LIN {X 0,Y 509.393,Z 1059.05,A -85,B 0,C 180,E1 -5481.271,E2 -5481.271} C_VEL
LIN {X 0,Y 509.308,Z 1064.075,A -85,B 0,C 180,E1 -5482.866,E2 -5482.866} C_VEL
LIN {X 0,Y 509.215,Z 1068.022,A -85,B 0,C 180,E1 -5484.456,E2 -5484.456} C_VEL
LIN {X 0,Y 509.196,Z 1070.928,A -85,B 0,C 180,E1 -5486.043,E2 -5486.043} C_VEL
LIN {X 0,Y 509.184,Z 1072.082,A -85,B 0,C 180,E1 -5486.835,E2 -5486.835} C_VEL
LIN {X 0,Y 509.107,Z 1073.515,A -85,B 0,C 180,E1 -5488.418,E2 -5488.418} C_VEL
LIN {X 0,Y 509.061,Z 1074,A -85,B 0,C 180,E1 -5490,E2 -5490} C_VEL
LIN {X 0,Y 509.107,Z 1073.515,A -85,B 0,C 180,E1 -5491.582,E2 -5491.582} C_VEL
LIN {X 0,Y 509.184,Z 1072.082,A -85,B 0,C 180,E1 -5493.165,E2 -5493.165} C_VEL
LIN {X 0,Y 509.142,Z 1069.669,A -85,B 0,C 180,E1 -5494.751,E2 -5494.751} C_VEL
LIN {X 0,Y 509.264,Z 1065.849,A -85,B 0,C 180,E1 -5496.476,E2 -5496.476} C_VEL
LIN {X 0,Y 509.332,Z 1061.713,A -85,B 0,C 180,E1 -5497.931,E2 -5497.931} C_VEL
LIN {X 0,Y 509.421,Z 1056.051,A -85,B 0,C 180,E1 -5499.529,E2 -5499.529} C_VEL
LIN {X 0,Y 509.628,Z 1051.052,A -85,B 0,C 180,E1 -5500.729,E2 -5500.729} C_VEL
LIN {X 0,Y 509.913,Z 1044.199,A -85,B 0,C 180,E1 -5502.133,E2 -5502.133} C_VEL
LIN {X 0,Y 510.2,Z 1036.178,A -85,B 0,C 180,E1 -5503.543,E2 -5503.543} C_VEL
LIN {X 0,Y 510.601,Z 1028.274,A -85,B 0,C 180,E1 -5504.752,E2 -5504.752} C_VEL
LIN {X 0,Y 511.042,Z 1019.227,A -85,B 0,C 180,E1 -5505.964,E2 -5505.964} C_VEL
LIN {X 0,Y 511.563,Z 1008.82,A -85,B 0,C 180,E1 -5507.179,E2 -5507.179} C_VEL
LIN {X 0,Y 512.103,Z 998.917,A -85,B 0,C 180,E1 -5508.192,E2 -5508.192} C_VEL
LIN {X 0,Y 512.69,Z 989.263,A -85,B 0,C 180,E1 -5509.065,E2 -5509.065} C_VEL
LIN {X 0,Y 513.308,Z 977.141,A -85,B 0,C 180,E1 -5510.016,E2 -5510.016} C_VEL
LIN {X 0,Y 513.876,Z 965.105,A -85,B 0,C 180,E1 -5510.829,E2 -5510.829} C_VEL
LIN {X 0,Y 514.531,Z 952.779,A -85,B 0,C 180,E1 -5511.535,E2 -5511.535} C_VEL
LIN {X 0,Y 515.092,Z 939.627,A -85,B 0,C 180,E1 -5512.169,E2 -5512.169} C_VEL
LIN {X 0,Y 515.587,Z 926.791,A -85,B 0,C 180,E1 -5512.674,E2 -5512.674} C_VEL
LIN {X 0,Y 515.947,Z 913.864,A -85,B 0,C 180,E1 -5513.081,E2 -5513.081} C_VEL
LIN {X 0,Y 516.291,Z 901.026,A -85,B 0,C 180,E1 -5513.383,E2 -5513.383} C_VEL
LIN {X 0,Y 516.696,Z 874.989,A -85,B 0,C 180,E1 -5513.789,E2 -5513.789} C_VEL
LIN {X 0,Y 518.063,Z 714.987,A -85,B 0,C 180,E1 -5516.115,E2 -5516.115} C_VEL
LIN {X 0,Y 513.214,Z 695.236,A -85,B 0,C 180,E1 -5516.696,E2 -5516.696} C_VEL
LIN {X 0,Y 514.044,Z 674.695,A -85,B 0,C 180,E1 -5519.709,E2 -5519.709} C_VEL
LIN {X 0,Y 513.889,Z 670.977,A -85,B 0,C 180,E1 -5520.284,E2 -5520.284} C_VEL
LIN {X 0,Y 509.916,Z 655.134,A -85,B 0,C 180,E1 -5523.033,E2 -5523.033} C_VEL
LIN {X 0,Y 509.867,Z 654.796,A -85,B 0,C 180,E1 -5523.178,E2 -5523.178} C_VEL
LIN {X 0,Y 509.83,Z 654.762,A -85,B 0,C 180,E1 -5526.352,E2 -5526.352} C_VEL
LIN {X 0,Y 509.83,Z 654.793,A -85,B 0,C 180,E1 -5529.47,E2 -5529.47} C_VEL
LIN {X 0,Y 509.842,Z 654.786,A -85,B 0,C 180,E1 -5532.487,E2 -5532.487} C_VEL
LIN {X 0,Y 509.85,Z 654.781,A -85,B 0,C 180,E1 -5535.331,E2 -5535.331} C_VEL
LIN {X 0,Y 509.866,Z 654.772,A -85,B 0,C 180,E1 -5538.576,E2 -5538.576} C_VEL
LIN {X 0,Y 509.849,Z 654.791,A -85,B 0,C 180,E1 -5541.785,E2 -5541.785} C_VEL
LIN {X 0,Y 509.839,Z 654.777,A -85,B 0,C 180,E1 -5544.623,E2 -5544.623} C_VEL
LIN {X 0,Y 509.858,Z 654.785,A -85,B 0,C 180,E1 -5547.481,E2 -5547.481} C_VEL
LIN {X 0,Y 509.873,Z 654.766,A -85,B 0,C 180,E1 -5550.268,E2 -5550.268} C_VEL
LIN {X 0,Y 509.878,Z 654.775,A -85,B 0,C 180,E1 -5552.944,E2 -5552.944} C_VEL
LIN {X 0,Y 509.86,Z 654.783,A -85,B 0,C 180,E1 -5555.573,E2 -5555.573} C_VEL
LIN {X 0,Y 509.813,Z 654.787,A -85,B 0,C 180,E1 -5558.148,E2 -5558.148} C_VEL
LIN {X 0,Y 509.855,Z 654.787,A -85,B 0,C 180,E1 -5560.681,E2 -5560.681} C_VEL
LIN {X 0,Y 509.877,Z 654.782,A -85,B 0,C 180,E1 -5563.174,E2 -5563.174} C_VEL
LIN {X 0,Y 509.854,Z 654.781,A -85,B 0,C 180,E1 -5565.634,E2 -5565.634} C_VEL
LIN {X 0,Y 509.919,Z 654.781,A -85,B 0,C 180,E1 -5568.875,E2 -5568.875} C_VEL
LIN {X 0,Y 509.941,Z 654.764,A -85,B 0,C 180,E1 -5572.078,E2 -5572.078} C_VEL
LIN {X 0,Y 510.001,Z 654.764,A -85,B 0,C 180,E1 -5574.464,E2 -5574.464} C_VEL
LIN {X 0,Y 510.045,Z 654.76,A -85,B 0,C 180,E1 -5577.631,E2 -5577.631} C_VEL
LIN {X 0,Y 510.056,Z 654.759,A -85,B 0,C 180,E1 -5580.789,E2 -5580.789} C_VEL
LIN {X 0,Y 509.95,Z 654.767,A -85,B 0,C 180,E1 -5583.16,E2 -5583.16} C_VEL
LIN {X 0,Y 509.972,Z 654.766,A -85,B 0,C 180,E1 -5586.329,E2 -5586.329} C_VEL
LIN {X 0,Y 509.908,Z 654.773,A -85,B 0,C 180,E1 -5588.72,E2 -5588.72} C_VEL
LIN {X 0,Y 509.893,Z 654.779,A -85,B 0,C 180,E1 -5591.932,E2 -5591.932} C_VEL
LIN {X 0,Y 509.882,Z 654.779,A -85,B 0,C 180,E1 -5595.242,E2 -5595.242} C_VEL
LIN {X 0,Y 509.877,Z 654.781,A -85,B 0,C 180,E1 -5598.001,E2 -5598.001} C_VEL
LIN {X 0,Y 509.848,Z 654.782,A -85,B 0,C 180,E1 -5601.001,E2 -5601.001} C_VEL
LIN {X 0,Y 509.841,Z 654.783,A -85,B 0,C 180,E1 -5603.563,E2 -5603.563} C_VEL
LIN {X 0,Y 509.902,Z 654.777,A -85,B 0,C 180,E1 -5606.379,E2 -5606.379} C_VEL
LIN {X 0,Y 509.875,Z 654.766,A -85,B 0,C 180,E1 -5608.844,E2 -5608.844} C_VEL
LIN {X 0,Y 509.816,Z 654.787,A -85,B 0,C 180,E1 -5611.59,E2 -5611.59} C_VEL
LIN {X 0,Y 509.845,Z 654.787,A -85,B 0,C 180,E1 -5614.413,E2 -5614.413} C_VEL
LIN {X 0,Y 509.809,Z 654.788,A -85,B 0,C 180,E1 -5617.341,E2 -5617.341} C_VEL
LIN {X 0,Y 509.854,Z 654.785,A -85,B 0,C 180,E1 -5620.38,E2 -5620.38} C_VEL
LIN {X 0,Y 509.833,Z 654.795,A -85,B 0,C 180,E1 -5623.065,E2 -5623.065} C_VEL
LIN {X 0,Y 509.822,Z 654.789,A -85,B 0,C 180,E1 -5625.793,E2 -5625.793} C_VEL
LIN {X 0,Y 509.857,Z 654.784,A -85,B 0,C 180,E1 -5628.576,E2 -5628.576} C_VEL
LIN {X 0,Y 509.844,Z 654.79,A -85,B 0,C 180,E1 -5631.787,E2 -5631.787} C_VEL
LIN {X 0,Y 509.825,Z 654.793,A -85,B 0,C 180,E1 -5633.744,E2 -5633.744} C_VEL
LIN {X 0,Y 509.159,Z 654.872,A -85,B 0,C 180,E1 -5634.404,E2 -5634.404} C_VEL
LIN {X 0,Y 506.341,Z 655.229,A -85,B 0,C 180,E1 -5635.476,E2 -5635.476} C_VEL
LIN {X 0,Y 503.947,Z 655.524,A -85,B 0,C 180,E1 -5636.339,E2 -5636.339} C_VEL
LIN {X 0,Y 502.899,Z 655.652,A -85,B 0,C 180,E1 -5637.006,E2 -5637.006} C_VEL
LIN {X 0,Y 502.802,Z 655.664,A -85,B 0,C 180,E1 -5637.231,E2 -5637.231} C_VEL
LIN {X 0,Y 502.824,Z 655.666,A -85,B 0,C 180,E1 -5640.062,E2 -5640.062} C_VEL
LIN {X 0,Y 502.828,Z 655.661,A -85,B 0,C 180,E1 -5642.534,E2 -5642.534} C_VEL
LIN {X 0,Y 502.823,Z 655.661,A -85,B 0,C 180,E1 -5645.299,E2 -5645.299} C_VEL
LIN {X 0,Y 502.78,Z 655.672,A -85,B 0,C 180,E1 -5647.827,E2 -5647.827} C_VEL
LIN {X 0,Y 502.82,Z 655.666,A -85,B 0,C 180,E1 -5650.401,E2 -5650.401} C_VEL
LIN {X 0,Y 502.829,Z 655.661,A -85,B 0,C 180,E1 -5652.932,E2 -5652.932} C_VEL
LIN {X 0,Y 502.841,Z 655.659,A -85,B 0,C 180,E1 -5655.429,E2 -5655.429} C_VEL
LIN {X 0,Y 502.873,Z 655.66,A -85,B 0,C 180,E1 -5658.717,E2 -5658.717} C_VEL
LIN {X 0,Y 502.898,Z 655.652,A -85,B 0,C 180,E1 -5661.967,E2 -5661.967} C_VEL
LIN {X 0,Y 502.934,Z 655.65,A -85,B 0,C 180,E1 -5664.387,E2 -5664.387} C_VEL
LIN {X 0,Y 503.021,Z 655.637,A -85,B 0,C 180,E1 -5667.598,E2 -5667.598} C_VEL
LIN {X 0,Y 503.024,Z 655.637,A -85,B 0,C 180,E1 -5670,E2 -5670} C_VEL
LIN {X 0,Y 503.021,Z 655.637,A -85,B 0,C 180,E1 -5672.402,E2 -5672.402} C_VEL
LIN {X 0,Y 502.934,Z 655.65,A -85,B 0,C 180,E1 -5675.613,E2 -5675.613} C_VEL
LIN {X 0,Y 502.898,Z 655.652,A -85,B 0,C 180,E1 -5678.033,E2 -5678.033} C_VEL
LIN {X 0,Y 502.873,Z 655.66,A -85,B 0,C 180,E1 -5681.283,E2 -5681.283} C_VEL
LIN {X 0,Y 502.841,Z 655.659,A -85,B 0,C 180,E1 -5684.571,E2 -5684.571} C_VEL
LIN {X 0,Y 502.857,Z 655.661,A -85,B 0,C 180,E1 -5687.907,E2 -5687.907} C_VEL
LIN {X 0,Y 502.823,Z 655.661,A -85,B 0,C 180,E1 -5690.536,E2 -5690.536} C_VEL
LIN {X 0,Y 502.792,Z 655.665,A -85,B 0,C 180,E1 -5693.04,E2 -5693.04} C_VEL
LIN {X 0,Y 502.835,Z 655.663,A -85,B 0,C 180,E1 -5695.675,E2 -5695.675} C_VEL
LIN {X 0,Y 502.836,Z 655.664,A -85,B 0,C 180,E1 -5698.372,E2 -5698.372} C_VEL
LIN {X 0,Y 502.791,Z 655.665,A -85,B 0,C 180,E1 -5701.499,E2 -5701.499} C_VEL
LIN {X 0,Y 502.799,Z 655.67,A -85,B 0,C 180,E1 -5704.444,E2 -5704.444} C_VEL
LIN {X 0,Y 502.774,Z 655.667,A -85,B 0,C 180,E1 -5707.178,E2 -5707.178} C_VEL
LIN {X 0,Y 502.814,Z 655.662,A -85,B 0,C 180,E1 -5710.011,E2 -5710.011} C_VEL
LIN {X 0,Y 502.764,Z 655.67,A -85,B 0,C 180,E1 -5713.231,E2 -5713.231} C_VEL
LIN {X 0,Y 502.781,Z 655.665,A -85,B 0,C 180,E1 -5715.661,E2 -5715.661} C_VEL
LIN {X 0,Y 502.83,Z 655.659,A -85,B 0,C 180,E1 -5717.865,E2 -5717.865} C_VEL
LIN {X 0,Y 502.812,Z 655.668,A -85,B 0,C 180,E1 -5721.026,E2 -5721.026} C_VEL
LIN {X 0,Y 502.775,Z 655.648,A -85,B 0,C 180,E1 -5724.167,E2 -5724.167} C_VEL
LIN {X 0,Y 502.823,Z 655.662,A -85,B 0,C 180,E1 -5726.993,E2 -5726.993} C_VEL
LIN {X 0,Y 502.82,Z 655.646,A -85,B 0,C 180,E1 -5730.061,E2 -5730.061} C_VEL
LIN {X 0,Y 502.825,Z 655.647,A -85,B 0,C 180,E1 -5732.533,E2 -5732.533} C_VEL
LIN {X 0,Y 502.82,Z 655.663,A -85,B 0,C 180,E1 -5735.298,E2 -5735.298} C_VEL
LIN {X 0,Y 502.809,Z 655.662,A -85,B 0,C 180,E1 -5737.828,E2 -5737.828} C_VEL
LIN {X 0,Y 502.814,Z 655.661,A -85,B 0,C 180,E1 -5740.4,E2 -5740.4} C_VEL
LIN {X 0,Y 502.825,Z 655.654,A -85,B 0,C 180,E1 -5742.932,E2 -5742.932} C_VEL
LIN {X 0,Y 502.834,Z 655.658,A -85,B 0,C 180,E1 -5745.429,E2 -5745.429} C_VEL
LIN {X 0,Y 502.87,Z 655.654,A -85,B 0,C 180,E1 -5748.717,E2 -5748.717} C_VEL
LIN {X 0,Y 502.891,Z 655.65,A -85,B 0,C 180,E1 -5751.967,E2 -5751.967} C_VEL
LIN {X 0,Y 502.952,Z 655.649,A -85,B 0,C 180,E1 -5754.387,E2 -5754.387} C_VEL
LIN {X 0,Y 503.015,Z 655.627,A -85,B 0,C 180,E1 -5757.598,E2 -5757.598} C_VEL
LIN {X 0,Y 503.015,Z 655.636,A -85,B 0,C 180,E1 -5760,E2 -5760} C_VEL
LIN {X 0,Y 503.015,Z 655.636,A -85,B 0,C 180,E1 -5762.402,E2 -5762.402} C_VEL
LIN {X 0,Y 502.952,Z 655.642,A -85,B 0,C 180,E1 -5765.614,E2 -5765.614} C_VEL
LIN {X 0,Y 502.892,Z 655.641,A -85,B 0,C 180,E1 -5768.034,E2 -5768.034} C_VEL
LIN {X 0,Y 502.887,Z 655.653,A -85,B 0,C 180,E1 -5771.283,E2 -5771.283} C_VEL
LIN {X 0,Y 502.834,Z 655.656,A -85,B 0,C 180,E1 -5774.571,E2 -5774.571} C_VEL
LIN {X 0,Y 502.852,Z 655.653,A -85,B 0,C 180,E1 -5777.907,E2 -5777.907} C_VEL
LIN {X 0,Y 502.818,Z 655.659,A -85,B 0,C 180,E1 -5780.537,E2 -5780.537} C_VEL
LIN {X 0,Y 502.787,Z 655.659,A -85,B 0,C 180,E1 -5783.041,E2 -5783.041} C_VEL
LIN {X 0,Y 502.832,Z 655.662,A -85,B 0,C 180,E1 -5785.676,E2 -5785.676} C_VEL
LIN {X 0,Y 502.833,Z 655.635,A -85,B 0,C 180,E1 -5788.373,E2 -5788.373} C_VEL
LIN {X 0,Y 502.789,Z 655.662,A -85,B 0,C 180,E1 -5791.5,E2 -5791.5} C_VEL
LIN {X 0,Y 502.799,Z 655.656,A -85,B 0,C 180,E1 -5794.446,E2 -5794.446} C_VEL
LIN {X 0,Y 502.774,Z 655.661,A -85,B 0,C 180,E1 -5797.179,E2 -5797.179} C_VEL
LIN {X 0,Y 502.828,Z 655.661,A -85,B 0,C 180,E1 -5800.011,E2 -5800.011} C_VEL
LIN {X 0,Y 502.82,Z 655.656,A -85,B 0,C 180,E1 -5802.203,E2 -5802.203} C_VEL
LIN {X 0,Y 502.794,Z 655.653,A -85,B 0,C 180,E1 -5805.469,E2 -5805.469} C_VEL
LIN {X 0,Y 502.824,Z 655.662,A -85,B 0,C 180,E1 -5807.865,E2 -5807.865} C_VEL
LIN {X 0,Y 502.797,Z 655.666,A -85,B 0,C 180,E1 -5811.025,E2 -5811.025} C_VEL
LIN {X 0,Y 502.78,Z 655.642,A -85,B 0,C 180,E1 -5814.168,E2 -5814.168} C_VEL
LIN {X 0,Y 502.851,Z 655.759,A -85,B 0,C 180,E1 -5816.559,E2 -5816.559} C_VEL
LIN {X 0,Y 506.42,Z 669.991,A -85,B 0,C 180,E1 -5819.105,E2 -5819.105} C_VEL
LIN {X 0,Y 507.298,Z 674.677,A -85,B 0,C 180,E1 -5819.886,E2 -5819.886} C_VEL
LIN {X 0,Y 506.412,Z 694.461,A -85,B 0,C 180,E1 -5822.866,E2 -5822.866} C_VEL
LIN {X 0,Y 506.693,Z 696.204,A -85,B 0,C 180,E1 -5822.965,E2 -5822.965} C_VEL
LIN {X 0,Y 511.701,Z 716.956,A -85,B 0,C 180,E1 -5823.569,E2 -5823.569} C_VEL
LIN {X 0,Y 509.898,Z 896.602,A -85,B 0,C 180,E1 -5826.225,E2 -5826.225} C_VEL
LIN {X 0,Y 509.497,Z 909.739,A -85,B 0,C 180,E1 -5826.502,E2 -5826.502} C_VEL
LIN {X 0,Y 509.137,Z 922.851,A -85,B 0,C 180,E1 -5826.888,E2 -5826.888} C_VEL
LIN {X 0,Y 508.613,Z 935.231,A -85,B 0,C 180,E1 -5827.346,E2 -5827.346} C_VEL
LIN {X 0,Y 508.097,Z 948.012,A -85,B 0,C 180,E1 -5827.932,E2 -5827.932} C_VEL
LIN {X 0,Y 507.494,Z 959.929,A -85,B 0,C 180,E1 -5828.581,E2 -5828.581} C_VEL
LIN {X 0,Y 506.819,Z 972.616,A -85,B 0,C 180,E1 -5829.399,E2 -5829.399} C_VEL
LIN {X 0,Y 506.202,Z 983.621,A -85,B 0,C 180,E1 -5830.22,E2 -5830.22} C_VEL
LIN {X 0,Y 505.486,Z 995.193,A -85,B 0,C 180,E1 -5831.215,E2 -5831.215} C_VEL
LIN {X 0,Y 504.949,Z 1004.935,A -85,B 0,C 180,E1 -5832.17,E2 -5832.17} C_VEL
LIN {X 0,Y 504.419,Z 1014.211,A -85,B 0,C 180,E1 -5833.196,E2 -5833.196} C_VEL
LIN {X 0,Y 503.865,Z 1023.624,A -85,B 0,C 180,E1 -5834.385,E2 -5834.385} C_VEL
LIN {X 0,Y 503.377,Z 1032.363,A -85,B 0,C 180,E1 -5835.652,E2 -5835.652} C_VEL
LIN {X 0,Y 502.964,Z 1040.89,A -85,B 0,C 180,E1 -5837.082,E2 -5837.082} C_VEL
LIN {X 0,Y 502.721,Z 1048.049,A -85,B 0,C 180,E1 -5838.475,E2 -5838.475} C_VEL
LIN {X 0,Y 502.431,Z 1054.443,A -85,B 0,C 180,E1 -5839.93,E2 -5839.93} C_VEL
LIN {X 0,Y 502.309,Z 1059.044,A -85,B 0,C 180,E1 -5841.147,E2 -5841.147} C_VEL
LIN {X 0,Y 502.231,Z 1064.071,A -85,B 0,C 180,E1 -5842.765,E2 -5842.765} C_VEL
LIN {X 0,Y 502.132,Z 1068.016,A -85,B 0,C 180,E1 -5844.378,E2 -5844.378} C_VEL
LIN {X 0,Y 502.09,Z 1070.924,A -85,B 0,C 180,E1 -5845.987,E2 -5845.987} C_VEL
LIN {X 0,Y 502.103,Z 1072.082,A -85,B 0,C 180,E1 -5846.791,E2 -5846.791} C_VEL
LIN {X 0,Y 502.03,Z 1073.518,A -85,B 0,C 180,E1 -5848.396,E2 -5848.396} C_VEL
LIN {X 0,Y 501.975,Z 1074,A -85,B 0,C 180,E1 -5850,E2 -5850} C_VEL
LIN {X 0,Y 502.03,Z 1073.518,A -85,B 0,C 180,E1 -5851.604,E2 -5851.604} C_VEL
LIN {X 0,Y 502.103,Z 1072.082,A -85,B 0,C 180,E1 -5853.209,E2 -5853.209} C_VEL
LIN {X 0,Y 502.061,Z 1069.666,A -85,B 0,C 180,E1 -5854.818,E2 -5854.818} C_VEL
LIN {X 0,Y 502.194,Z 1065.145,A -85,B 0,C 180,E1 -5856.831,E2 -5856.831} C_VEL
LIN {X 0,Y 502.248,Z 1061.707,A -85,B 0,C 180,E1 -5858.044,E2 -5858.044} C_VEL
LIN {X 0,Y 502.354,Z 1056.046,A -85,B 0,C 180,E1 -5859.664,E2 -5859.664} C_VEL
LIN {X 0,Y 502.585,Z 1051.046,A -85,B 0,C 180,E1 -5860.881,E2 -5860.881} C_VEL
LIN {X 0,Y 502.878,Z 1044.193,A -85,B 0,C 180,E1 -5862.305,E2 -5862.305} C_VEL
LIN {X 0,Y 503.2,Z 1036.171,A -85,B 0,C 180,E1 -5863.735,E2 -5863.735} C_VEL
LIN {X 0,Y 503.67,Z 1028.267,A -85,B 0,C 180,E1 -5864.959,E2 -5864.959} C_VEL
LIN {X 0,Y 504.152,Z 1019.22,A -85,B 0,C 180,E1 -5866.188,E2 -5866.188} C_VEL
LIN {X 0,Y 504.599,Z 1010.657,A -85,B 0,C 180,E1 -5867.215,E2 -5867.215} C_VEL
LIN {X 0,Y 505.266,Z 998.783,A -85,B 0,C 180,E1 -5868.447,E2 -5868.447} C_VEL
LIN {X 0,Y 505.944,Z 988.463,A -85,B 0,C 180,E1 -5869.381,E2 -5869.381} C_VEL
LIN {X 0,Y 506.575,Z 976.934,A -85,B 0,C 180,E1 -5870.294,E2 -5870.294} C_VEL
LIN {X 0,Y 507.177,Z 964.897,A -85,B 0,C 180,E1 -5871.117,E2 -5871.117} C_VEL
LIN {X 0,Y 507.851,Z 953.134,A -85,B 0,C 180,E1 -5871.803,E2 -5871.803} C_VEL
LIN {X 0,Y 508.465,Z 939.42,A -85,B 0,C 180,E1 -5872.473,E2 -5872.473} C_VEL
LIN {X 0,Y 509.013,Z 926.584,A -85,B 0,C 180,E1 -5872.984,E2 -5872.984} C_VEL
LIN {X 0,Y 509.39,Z 913.658,A -85,B 0,C 180,E1 -5873.396,E2 -5873.396} C_VEL
LIN {X 0,Y 509.765,Z 900.82,A -85,B 0,C 180,E1 -5873.701,E2 -5873.701} C_VEL
LIN {X 0,Y 510.216,Z 874.784,A -85,B 0,C 180,E1 -5874.11,E2 -5874.11} C_VEL
LIN {X 0,Y 511.593,Z 715.983,A -85,B 0,C 180,E1 -5876.452,E2 -5876.452} C_VEL
LIN {X 0,Y 506.442,Z 694.904,A -85,B 0,C 180,E1 -5877.087,E2 -5877.087} C_VEL
LIN {X 0,Y 507.301,Z 675.964,A -85,B 0,C 180,E1 -5879.915,E2 -5879.915} C_VEL
LIN {X 0,Y 506.98,Z 672.28,A -85,B 0,C 180,E1 -5880.504,E2 -5880.504} C_VEL
LIN {X 0,Y 502.881,Z 655.971,A -85,B 0,C 180,E1 -5883.385,E2 -5883.385} C_VEL
LIN {X 0,Y 502.823,Z 655.687,A -85,B 0,C 180,E1 -5883.509,E2 -5883.509} C_VEL
LIN {X 0,Y 502.778,Z 655.641,A -85,B 0,C 180,E1 -5885.95,E2 -5885.95} C_VEL
LIN {X 0,Y 502.797,Z 655.666,A -85,B 0,C 180,E1 -5888.975,E2 -5888.975} C_VEL
LIN {X 0,Y 502.824,Z 655.662,A -85,B 0,C 180,E1 -5892.135,E2 -5892.135} C_VEL
LIN {X 0,Y 502.795,Z 655.662,A -85,B 0,C 180,E1 -5895.467,E2 -5895.467} C_VEL
LIN {X 0,Y 502.832,Z 655.654,A -85,B 0,C 180,E1 -5897.864,E2 -5897.864} C_VEL
LIN {X 0,Y 502.815,Z 655.661,A -85,B 0,C 180,E1 -5901.025,E2 -5901.025} C_VEL
LIN {X 0,Y 502.778,Z 655.656,A -85,B 0,C 180,E1 -5904.166,E2 -5904.166} C_VEL
LIN {X 0,Y 502.825,Z 655.659,A -85,B 0,C 180,E1 -5906.992,E2 -5906.992} C_VEL
LIN {X 0,Y 502.822,Z 655.647,A -85,B 0,C 180,E1 -5910.061,E2 -5910.061} C_VEL
LIN {X 0,Y 502.826,Z 655.651,A -85,B 0,C 180,E1 -5912.533,E2 -5912.533} C_VEL
LIN {X 0,Y 502.819,Z 655.66,A -85,B 0,C 180,E1 -5915.298,E2 -5915.298} C_VEL
LIN {X 0,Y 502.775,Z 655.66,A -85,B 0,C 180,E1 -5917.826,E2 -5917.826} C_VEL
LIN {X 0,Y 502.816,Z 655.667,A -85,B 0,C 180,E1 -5920.4,E2 -5920.4} C_VEL
LIN {X 0,Y 502.827,Z 655.663,A -85,B 0,C 180,E1 -5922.931,E2 -5922.931} C_VEL
LIN {X 0,Y 502.834,Z 655.657,A -85,B 0,C 180,E1 -5925.429,E2 -5925.429} C_VEL
LIN {X 0,Y 502.887,Z 655.654,A -85,B 0,C 180,E1 -5928.717,E2 -5928.717} C_VEL
LIN {X 0,Y 502.892,Z 655.641,A -85,B 0,C 180,E1 -5931.966,E2 -5931.966} C_VEL
LIN {X 0,Y 502.952,Z 655.642,A -85,B 0,C 180,E1 -5934.386,E2 -5934.386} C_VEL
LIN {X 0,Y 503.015,Z 655.636,A -85,B 0,C 180,E1 -5937.598,E2 -5937.598} C_VEL
LIN {X 0,Y 503.015,Z 655.635,A -85,B 0,C 180,E1 -5940,E2 -5940} C_VEL
LIN {X 0,Y 503.015,Z 655.626,A -85,B 0,C 180,E1 -5942.402,E2 -5942.402} C_VEL
LIN {X 0,Y 502.952,Z 655.65,A -85,B 0,C 180,E1 -5945.613,E2 -5945.613} C_VEL
LIN {X 0,Y 502.891,Z 655.651,A -85,B 0,C 180,E1 -5948.033,E2 -5948.033} C_VEL
LIN {X 0,Y 502.87,Z 655.654,A -85,B 0,C 180,E1 -5951.283,E2 -5951.283} C_VEL
LIN {X 0,Y 502.834,Z 655.658,A -85,B 0,C 180,E1 -5954.571,E2 -5954.571} C_VEL
LIN {X 0,Y 502.85,Z 655.655,A -85,B 0,C 180,E1 -5957.907,E2 -5957.907} C_VEL
LIN {X 0,Y 502.819,Z 655.662,A -85,B 0,C 180,E1 -5960.537,E2 -5960.537} C_VEL
LIN {X 0,Y 502.804,Z 655.66,A -85,B 0,C 180,E1 -5963.04,E2 -5963.04} C_VEL
LIN {X 0,Y 502.831,Z 655.658,A -85,B 0,C 180,E1 -5965.676,E2 -5965.676} C_VEL
LIN {X 0,Y 502.832,Z 655.642,A -85,B 0,C 180,E1 -5968.373,E2 -5968.373} C_VEL
LIN {X 0,Y 502.786,Z 655.663,A -85,B 0,C 180,E1 -5971.5,E2 -5971.5} C_VEL
LIN {X 0,Y 502.797,Z 655.663,A -85,B 0,C 180,E1 -5974.445,E2 -5974.445} C_VEL
LIN {X 0,Y 502.771,Z 655.66,A -85,B 0,C 180,E1 -5977.179,E2 -5977.179} C_VEL
LIN {X 0,Y 502.818,Z 655.66,A -85,B 0,C 180,E1 -5980.012,E2 -5980.012} C_VEL
LIN {X 0,Y 502.818,Z 655.661,A -85,B 0,C 180,E1 -5982.203,E2 -5982.203} C_VEL
LIN {X 0,Y 502.792,Z 655.669,A -85,B 0,C 180,E1 -5985.469,E2 -5985.469} C_VEL
LIN {X 0,Y 502.818,Z 655.665,A -85,B 0,C 180,E1 -5989.004,E2 -5989.004} C_VEL
LIN {X 0,Y 502.787,Z 655.666,A -85,B 0,C 180,E1 -5992.047,E2 -5992.047} C_VEL
LIN {X 0,Y 502.802,Z 655.664,A -85,B 0,C 180,E1 -5995.036,E2 -5995.036} C_VEL
LIN {X 0,Y 502.802,Z 655.664,A -85,B 0,C 180,E1 -5997.231,E2 -5997.231} C_VEL
LIN {X 0,Y 502.105,Z 655.755,A -85,B 0,C 180,E1 -5997.9,E2 -5997.9} C_VEL
LIN {X 0,Y 499.246,Z 656.107,A -85,B 0,C 180,E1 -5998.986,E2 -5998.986} C_VEL
LIN {X 0,Y 496.855,Z 656.41,A -85,B 0,C 180,E1 -5999.861,E2 -5999.861} C_VEL
LIN {X 0,Y 495.837,Z 656.532,A -85,B 0,C 180,E1 -6000.537,E2 -6000.537} C_VEL
LIN {X 0,Y 495.757,Z 656.541,A -85,B 0,C 180,E1 -6000.765,E2 -6000.765} C_VEL
LIN {X 0,Y 495.785,Z 656.543,A -85,B 0,C 180,E1 -6003.933,E2 -6003.933} C_VEL
LIN {X 0,Y 495.76,Z 656.541,A -85,B 0,C 180,E1 -6007.138,E2 -6007.138} C_VEL
LIN {X 0,Y 495.767,Z 656.546,A -85,B 0,C 180,E1 -6010.11,E2 -6010.11} C_VEL
LIN {X 0,Y 495.782,Z 656.541,A -85,B 0,C 180,E1 -6012.682,E2 -6012.682} C_VEL
LIN {X 0,Y 495.786,Z 656.539,A -85,B 0,C 180,E1 -6015.217,E2 -6015.217} C_VEL
LIN {X 0,Y 495.847,Z 656.535,A -85,B 0,C 180,E1 -6018.555,E2 -6018.555} C_VEL
LIN {X 0,Y 495.869,Z 656.528,A -85,B 0,C 180,E1 -6021.852,E2 -6021.852} C_VEL
LIN {X 0,Y 495.892,Z 656.527,A -85,B 0,C 180,E1 -6024.307,E2 -6024.307} C_VEL
LIN {X 0,Y 495.99,Z 656.513,A -85,B 0,C 180,E1 -6027.564,E2 -6027.564} C_VEL
LIN {X 0,Y 495.995,Z 656.512,A -85,B 0,C 180,E1 -6030,E2 -6030} C_VEL
LIN {X 0,Y 495.99,Z 656.513,A -85,B 0,C 180,E1 -6032.436,E2 -6032.436} C_VEL
LIN {X 0,Y 495.892,Z 656.527,A -85,B 0,C 180,E1 -6035.693,E2 -6035.693} C_VEL
LIN {X 0,Y 495.869,Z 656.528,A -85,B 0,C 180,E1 -6038.148,E2 -6038.148} C_VEL
LIN {X 0,Y 495.847,Z 656.535,A -85,B 0,C 180,E1 -6041.445,E2 -6041.445} C_VEL
LIN {X 0,Y 495.786,Z 656.539,A -85,B 0,C 180,E1 -6044.783,E2 -6044.783} C_VEL
LIN {X 0,Y 495.782,Z 656.541,A -85,B 0,C 180,E1 -6047.318,E2 -6047.318} C_VEL
LIN {X 0,Y 495.767,Z 656.546,A -85,B 0,C 180,E1 -6049.89,E2 -6049.89} C_VEL
LIN {X 0,Y 495.76,Z 656.541,A -85,B 0,C 180,E1 -6052.862,E2 -6052.862} C_VEL
LIN {X 0,Y 495.785,Z 656.543,A -85,B 0,C 180,E1 -6056.067,E2 -6056.067} C_VEL
LIN {X 0,Y 495.774,Z 656.54,A -85,B 0,C 180,E1 -6058.814,E2 -6058.814} C_VEL
LIN {X 0,Y 495.753,Z 656.543,A -85,B 0,C 180,E1 -6061.726,E2 -6061.726} C_VEL
LIN {X 0,Y 495.769,Z 656.544,A -85,B 0,C 180,E1 -6064.695,E2 -6064.695} C_VEL
LIN {X 0,Y 495.724,Z 656.545,A -85,B 0,C 180,E1 -6067.561,E2 -6067.561} C_VEL
LIN {X 0,Y 495.772,Z 656.545,A -85,B 0,C 180,E1 -6070.698,E2 -6070.698} C_VEL
LIN {X 0,Y 495.725,Z 656.544,A -85,B 0,C 180,E1 -6074,E2 -6074} C_VEL
LIN {X 0,Y 495.756,Z 656.546,A -85,B 0,C 180,E1 -6077.121,E2 -6077.121} C_VEL
LIN {X 0,Y 495.782,Z 656.538,A -85,B 0,C 180,E1 -6080.365,E2 -6080.365} C_VEL
LIN {X 0,Y 495.724,Z 656.528,A -85,B 0,C 180,E1 -6083.456,E2 -6083.456} C_VEL
LIN {X 0,Y 495.751,Z 656.539,A -85,B 0,C 180,E1 -6086.436,E2 -6086.436} C_VEL
LIN {X 0,Y 495.747,Z 656.537,A -85,B 0,C 180,E1 -6089.313,E2 -6089.313} C_VEL
LIN {X 0,Y 495.772,Z 656.525,A -85,B 0,C 180,E1 -6092.109,E2 -6092.109} C_VEL
LIN {X 0,Y 495.779,Z 656.536,A -85,B 0,C 180,E1 -6094.833,E2 -6094.833} C_VEL
LIN {X 0,Y 495.772,Z 656.539,A -85,B 0,C 180,E1 -6097.496,E2 -6097.496} C_VEL
LIN {X 0,Y 495.767,Z 656.542,A -85,B 0,C 180,E1 -6100.11,E2 -6100.11} C_VEL
LIN {X 0,Y 495.776,Z 656.532,A -85,B 0,C 180,E1 -6102.681,E2 -6102.681} C_VEL
LIN {X 0,Y 495.779,Z 656.536,A -85,B 0,C 180,E1 -6105.217,E2 -6105.217} C_VEL
LIN {X 0,Y 495.844,Z 656.531,A -85,B 0,C 180,E1 -6108.555,E2 -6108.555} C_VEL
LIN {X 0,Y 495.863,Z 656.524,A -85,B 0,C 180,E1 -6111.852,E2 -6111.852} C_VEL
LIN {X 0,Y 495.906,Z 656.525,A -85,B 0,C 180,E1 -6114.307,E2 -6114.307} C_VEL
LIN {X 0,Y 495.984,Z 656.502,A -85,B 0,C 180,E1 -6117.564,E2 -6117.564} C_VEL
LIN {X 0,Y 495.986,Z 656.512,A -85,B 0,C 180,E1 -6120,E2 -6120} C_VEL
LIN {X 0,Y 495.984,Z 656.511,A -85,B 0,C 180,E1 -6122.437,E2 -6122.437} C_VEL
LIN {X 0,Y 495.907,Z 656.52,A -85,B 0,C 180,E1 -6125.694,E2 -6125.694} C_VEL
LIN {X 0,Y 495.863,Z 656.516,A -85,B 0,C 180,E1 -6128.148,E2 -6128.148} C_VEL
LIN {X 0,Y 495.861,Z 656.526,A -85,B 0,C 180,E1 -6131.445,E2 -6131.445} C_VEL
LIN {X 0,Y 495.779,Z 656.536,A -85,B 0,C 180,E1 -6134.783,E2 -6134.783} C_VEL
LIN {X 0,Y 495.778,Z 656.537,A -85,B 0,C 180,E1 -6137.319,E2 -6137.319} C_VEL
LIN {X 0,Y 495.768,Z 656.541,A -85,B 0,C 180,E1 -6139.891,E2 -6139.891} C_VEL
LIN {X 0,Y 495.756,Z 656.534,A -85,B 0,C 180,E1 -6142.863,E2 -6142.863} C_VEL
LIN {X 0,Y 495.79,Z 656.533,A -85,B 0,C 180,E1 -6146.068,E2 -6146.068} C_VEL
LIN {X 0,Y 495.771,Z 656.512,A -85,B 0,C 180,E1 -6148.815,E2 -6148.815} C_VEL
LIN {X 0,Y 495.751,Z 656.542,A -85,B 0,C 180,E1 -6151.727,E2 -6151.727} C_VEL
LIN {X 0,Y 495.769,Z 656.529,A -85,B 0,C 180,E1 -6154.696,E2 -6154.696} C_VEL
LIN {X 0,Y 495.726,Z 656.541,A -85,B 0,C 180,E1 -6157.562,E2 -6157.562} C_VEL
LIN {X 0,Y 495.794,Z 656.535,A -85,B 0,C 180,E1 -6160.054,E2 -6160.054} C_VEL
LIN {X 0,Y 495.758,Z 656.543,A -85,B 0,C 180,E1 -6162.88,E2 -6162.88} C_VEL
LIN {X 0,Y 495.73,Z 656.535,A -85,B 0,C 180,E1 -6166,E2 -6166} C_VEL
LIN {X 0,Y 495.758,Z 656.538,A -85,B 0,C 180,E1 -6168.707,E2 -6168.707} C_VEL
LIN {X 0,Y 495.746,Z 656.54,A -85,B 0,C 180,E1 -6171.409,E2 -6171.409} C_VEL
LIN {X 0,Y 495.753,Z 656.52,A -85,B 0,C 180,E1 -6174.464,E2 -6174.464} C_VEL
LIN {X 0,Y 495.798,Z 656.619,A -85,B 0,C 180,E1 -6176.196,E2 -6176.196} C_VEL
LIN {X 0,Y 499.085,Z 669.753,A -85,B 0,C 180,E1 -6178.6,E2 -6178.6} C_VEL
LIN {X 0,Y 500.481,Z 675.745,A -85,B 0,C 180,E1 -6179.634,E2 -6179.634} C_VEL
LIN {X 0,Y 499.756,Z 691.891,A -85,B 0,C 180,E1 -6182.123,E2 -6182.123} C_VEL
LIN {X 0,Y 499.664,Z 694.758,A -85,B 0,C 180,E1 -6182.519,E2 -6182.519} C_VEL
LIN {X 0,Y 505.261,Z 717.615,A -85,B 0,C 180,E1 -6183.219,E2 -6183.219} C_VEL
LIN {X 0,Y 503.5,Z 892.178,A -85,B 0,C 180,E1 -6185.822,E2 -6185.822} C_VEL
LIN {X 0,Y 503.076,Z 907.575,A -85,B 0,C 180,E1 -6186.129,E2 -6186.129} C_VEL
LIN {X 0,Y 502.661,Z 921.153,A -85,B 0,C 180,E1 -6186.518,E2 -6186.518} C_VEL
LIN {X 0,Y 502.056,Z 935.025,A -85,B 0,C 180,E1 -6187.033,E2 -6187.033} C_VEL
LIN {X 0,Y 501.479,Z 947.613,A -85,B 0,C 180,E1 -6187.615,E2 -6187.615} C_VEL
LIN {X 0,Y 500.821,Z 960.031,A -85,B 0,C 180,E1 -6188.301,E2 -6188.301} C_VEL
LIN {X 0,Y 500.207,Z 970.97,A -85,B 0,C 180,E1 -6189.006,E2 -6189.006} C_VEL
LIN {X 0,Y 499.423,Z 983.413,A -85,B 0,C 180,E1 -6189.94,E2 -6189.94} C_VEL
LIN {X 0,Y 498.724,Z 994.276,A -85,B 0,C 180,E1 -6190.881,E2 -6190.881} C_VEL
LIN {X 0,Y 498.098,Z 1004.727,A -85,B 0,C 180,E1 -6191.916,E2 -6191.916} C_VEL
LIN {X 0,Y 497.504,Z 1014.002,A -85,B 0,C 180,E1 -6192.955,E2 -6192.955} C_VEL
LIN {X 0,Y 496.873,Z 1024.015,A -85,B 0,C 180,E1 -6194.24,E2 -6194.24} C_VEL
LIN {X 0,Y 496.424,Z 1032.265,A -85,B 0,C 180,E1 -6195.446,E2 -6195.446} C_VEL
LIN {X 0,Y 495.962,Z 1040.865,A -85,B 0,C 180,E1 -6196.896,E2 -6196.896} C_VEL
LIN {X 0,Y 495.726,Z 1047.393,A -85,B 0,C 180,E1 -6198.168,E2 -6198.168} C_VEL
LIN {X 0,Y 495.383,Z 1054.439,A -85,B 0,C 180,E1 -6199.786,E2 -6199.786} C_VEL
LIN {X 0,Y 495.237,Z 1059.037,A -85,B 0,C 180,E1 -6201.019,E2 -6201.019} C_VEL
LIN {X 0,Y 495.15,Z 1064.067,A -85,B 0,C 180,E1 -6202.661,E2 -6202.661} C_VEL
LIN {X 0,Y 495.053,Z 1068.011,A -85,B 0,C 180,E1 -6204.297,E2 -6204.297} C_VEL
LIN {X 0,Y 494.985,Z 1070.919,A -85,B 0,C 180,E1 -6205.929,E2 -6205.929} C_VEL
LIN {X 0,Y 495.023,Z 1072.081,A -85,B 0,C 180,E1 -6206.745,E2 -6206.745} C_VEL
LIN {X 0,Y 494.956,Z 1073.521,A -85,B 0,C 180,E1 -6208.373,E2 -6208.373} C_VEL
LIN {X 0,Y 494.893,Z 1074,A -85,B 0,C 180,E1 -6210,E2 -6210} C_VEL
LIN {X 0,Y 494.956,Z 1073.521,A -85,B 0,C 180,E1 -6211.627,E2 -6211.627} C_VEL
LIN {X 0,Y 495.023,Z 1072.081,A -85,B 0,C 180,E1 -6213.255,E2 -6213.255} C_VEL
LIN {X 0,Y 494.984,Z 1069.66,A -85,B 0,C 180,E1 -6214.887,E2 -6214.887} C_VEL
LIN {X 0,Y 495.102,Z 1066.213,A -85,B 0,C 180,E1 -6216.52,E2 -6216.52} C_VEL
LIN {X 0,Y 495.183,Z 1061.701,A -85,B 0,C 180,E1 -6218.159,E2 -6218.159} C_VEL
LIN {X 0,Y 495.291,Z 1056.042,A -85,B 0,C 180,E1 -6219.804,E2 -6219.804} C_VEL
LIN {X 0,Y 495.55,Z 1051.039,A -85,B 0,C 180,E1 -6221.038,E2 -6221.038} C_VEL
LIN {X 0,Y 495.84,Z 1044.188,A -85,B 0,C 180,E1 -6222.483,E2 -6222.483} C_VEL
LIN {X 0,Y 496.212,Z 1036.105,A -85,B 0,C 180,E1 -6223.932,E2 -6223.932} C_VEL
LIN {X 0,Y 496.721,Z 1028.138,A -85,B 0,C 180,E1 -6225.174,E2 -6225.174} C_VEL
LIN {X 0,Y 497.212,Z 1019.021,A -85,B 0,C 180,E1 -6226.421,E2 -6226.421} C_VEL
LIN {X 0,Y 497.708,Z 1010.448,A -85,B 0,C 180,E1 -6227.461,E2 -6227.461} C_VEL
LIN {X 0,Y 498.461,Z 998.576,A -85,B 0,C 180,E1 -6228.708,E2 -6228.708} C_VEL
LIN {X 0,Y 499.143,Z 988.493,A -85,B 0,C 180,E1 -6229.635,E2 -6229.635} C_VEL
LIN {X 0,Y 499.847,Z 976.726,A -85,B 0,C 180,E1 -6230.579,E2 -6230.579} C_VEL
LIN {X 0,Y 500.51,Z 964.69,A -85,B 0,C 180,E1 -6231.412,E2 -6231.412} C_VEL
LIN {X 0,Y 501.248,Z 952.514,A -85,B 0,C 180,E1 -6232.128,E2 -6232.128} C_VEL
LIN {X 0,Y 501.863,Z 939.213,A -85,B 0,C 180,E1 -6232.786,E2 -6232.786} C_VEL
LIN {X 0,Y 502.453,Z 926.378,A -85,B 0,C 180,E1 -6233.301,E2 -6233.301} C_VEL
LIN {X 0,Y 502.877,Z 913.452,A -85,B 0,C 180,E1 -6233.717,E2 -6233.717} C_VEL
LIN {X 0,Y 503.249,Z 900.614,A -85,B 0,C 180,E1 -6234.027,E2 -6234.027} C_VEL
LIN {X 0,Y 503.731,Z 874.578,A -85,B 0,C 180,E1 -6234.441,E2 -6234.441} C_VEL
LIN {X 0,Y 505.295,Z 717.582,A -85,B 0,C 180,E1 -6236.78,E2 -6236.78} C_VEL
LIN {X 0,Y 499.686,Z 694.533,A -85,B 0,C 180,E1 -6237.494,E2 -6237.494} C_VEL
LIN {X 0,Y 500.571,Z 677.234,A -85,B 0,C 180,E1 -6240.127,E2 -6240.127} C_VEL
LIN {X 0,Y 500.023,Z 673.565,A -85,B 0,C 180,E1 -6240.737,E2 -6240.737} C_VEL
LIN {X 0,Y 496.056,Z 657.839,A -85,B 0,C 180,E1 -6243.541,E2 -6243.541} C_VEL
LIN {X 0,Y 495.776,Z 656.584,A -85,B 0,C 180,E1 -6243.837,E2 -6243.837} C_VEL
LIN {X 0,Y 495.728,Z 656.514,A -85,B 0,C 180,E1 -6246.543,E2 -6246.543} C_VEL
LIN {X 0,Y 495.752,Z 656.545,A -85,B 0,C 180,E1 -6249.637,E2 -6249.637} C_VEL
LIN {X 0,Y 495.735,Z 656.544,A -85,B 0,C 180,E1 -6252.507,E2 -6252.507} C_VEL
LIN {X 0,Y 495.743,Z 656.535,A -85,B 0,C 180,E1 -6255.139,E2 -6255.139} C_VEL
LIN {X 0,Y 495.779,Z 656.528,A -85,B 0,C 180,E1 -6258.221,E2 -6258.221} C_VEL
LIN {X 0,Y 495.771,Z 656.54,A -85,B 0,C 180,E1 -6261.229,E2 -6261.229} C_VEL
LIN {X 0,Y 495.75,Z 656.531,A -85,B 0,C 180,E1 -6264.463,E2 -6264.463} C_VEL
LIN {X 0,Y 495.761,Z 656.54,A -85,B 0,C 180,E1 -6267.405,E2 -6267.405} C_VEL
LIN {X 0,Y 495.773,Z 656.52,A -85,B 0,C 180,E1 -6270.254,E2 -6270.254} C_VEL
LIN {X 0,Y 495.825,Z 656.524,A -85,B 0,C 180,E1 -6273.248,E2 -6273.248} C_VEL
LIN {X 0,Y 495.743,Z 656.542,A -85,B 0,C 180,E1 -6275.724,E2 -6275.724} C_VEL
LIN {X 0,Y 495.734,Z 656.543,A -85,B 0,C 180,E1 -6278.371,E2 -6278.371} C_VEL
LIN {X 0,Y 495.775,Z 656.536,A -85,B 0,C 180,E1 -6280.971,E2 -6280.971} C_VEL
LIN {X 0,Y 495.771,Z 656.537,A -85,B 0,C 180,E1 -6283.53,E2 -6283.53} C_VEL
LIN {X 0,Y 495.786,Z 656.534,A -85,B 0,C 180,E1 -6286.055,E2 -6286.055} C_VEL
LIN {X 0,Y 495.861,Z 656.526,A -85,B 0,C 180,E1 -6288.555,E2 -6288.555} C_VEL
LIN {X 0,Y 495.863,Z 656.517,A -85,B 0,C 180,E1 -6291.852,E2 -6291.852} C_VEL
LIN {X 0,Y 495.907,Z 656.519,A -85,B 0,C 180,E1 -6294.306,E2 -6294.306} C_VEL
LIN {X 0,Y 495.984,Z 656.511,A -85,B 0,C 180,E1 -6297.563,E2 -6297.563} C_VEL
LIN {X 0,Y 495.986,Z 656.511,A -85,B 0,C 180,E1 -6300,E2 -6300} C_VEL
LIN {X 0,Y 495.984,Z 656.502,A -85,B 0,C 180,E1 -6302.436,E2 -6302.436} C_VEL
LIN {X 0,Y 495.906,Z 656.526,A -85,B 0,C 180,E1 -6305.693,E2 -6305.693} C_VEL
LIN {X 0,Y 495.863,Z 656.525,A -85,B 0,C 180,E1 -6308.148,E2 -6308.148} C_VEL
LIN {X 0,Y 495.844,Z 656.532,A -85,B 0,C 180,E1 -6311.445,E2 -6311.445} C_VEL
LIN {X 0,Y 495.779,Z 656.536,A -85,B 0,C 180,E1 -6314.783,E2 -6314.783} C_VEL
LIN {X 0,Y 495.776,Z 656.533,A -85,B 0,C 180,E1 -6317.319,E2 -6317.319} C_VEL
LIN {X 0,Y 495.767,Z 656.542,A -85,B 0,C 180,E1 -6319.89,E2 -6319.89} C_VEL
LIN {X 0,Y 495.776,Z 656.536,A -85,B 0,C 180,E1 -6322.869,E2 -6322.869} C_VEL
LIN {X 0,Y 495.79,Z 656.539,A -85,B 0,C 180,E1 -6326.067,E2 -6326.067} C_VEL
LIN {X 0,Y 495.769,Z 656.519,A -85,B 0,C 180,E1 -6328.814,E2 -6328.814} C_VEL
LIN {X 0,Y 495.749,Z 656.539,A -85,B 0,C 180,E1 -6331.726,E2 -6331.726} C_VEL
LIN {X 0,Y 495.767,Z 656.532,A -85,B 0,C 180,E1 -6334.696,E2 -6334.696} C_VEL
LIN {X 0,Y 495.723,Z 656.54,A -85,B 0,C 180,E1 -6337.562,E2 -6337.562} C_VEL
LIN {X 0,Y 495.785,Z 656.536,A -85,B 0,C 180,E1 -6340.052,E2 -6340.052} C_VEL
LIN {X 0,Y 495.756,Z 656.546,A -85,B 0,C 180,E1 -6342.879,E2 -6342.879} C_VEL
LIN {X 0,Y 495.725,Z 656.544,A -85,B 0,C 180,E1 -6346,E2 -6346} C_VEL
LIN {X 0,Y 495.772,Z 656.545,A -85,B 0,C 180,E1 -6349.302,E2 -6349.302} C_VEL
LIN {X 0,Y 495.724,Z 656.545,A -85,B 0,C 180,E1 -6352.439,E2 -6352.439} C_VEL
LIN {X 0,Y 495.778,Z 656.545,A -85,B 0,C 180,E1 -6355.458,E2 -6355.458} C_VEL
LIN {X 0,Y 495.753,Z 656.542,A -85,B 0,C 180,E1 -6358.365,E2 -6358.365} C_VEL
LIN {X 0,Y 495.757,Z 656.541,A -85,B 0,C 180,E1 -6360.765,E2 -6360.765} C_VEL
LIN {X 0,Y 495.096,Z 656.627,A -85,B 0,C 180,E1 -6361.444,E2 -6361.444} C_VEL
LIN {X 0,Y 492.235,Z 656.981,A -85,B 0,C 180,E1 -6362.547,E2 -6362.547} C_VEL
LIN {X 0,Y 489.825,Z 657.283,A -85,B 0,C 180,E1 -6363.435,E2 -6363.435} C_VEL
LIN {X 0,Y 488.809,Z 657.412,A -85,B 0,C 180,E1 -6364.122,E2 -6364.122} C_VEL
LIN {X 0,Y 488.737,Z 657.418,A -85,B 0,C 180,E1 -6364.354,E2 -6364.354} C_VEL
LIN {X 0,Y 488.723,Z 657.418,A -85,B 0,C 180,E1 -6367.154,E2 -6367.154} C_VEL
LIN {X 0,Y 488.72,Z 657.421,A -85,B 0,C 180,E1 -6369.811,E2 -6369.811} C_VEL
LIN {X 0,Y 488.729,Z 657.422,A -85,B 0,C 180,E1 -6372.424,E2 -6372.424} C_VEL
LIN {X 0,Y 488.757,Z 657.416,A -85,B 0,C 180,E1 -6375,E2 -6375} C_VEL
LIN {X 0,Y 488.801,Z 657.413,A -85,B 0,C 180,E1 -6378.388,E2 -6378.388} C_VEL
LIN {X 0,Y 488.814,Z 657.407,A -85,B 0,C 180,E1 -6381.734,E2 -6381.734} C_VEL
LIN {X 0,Y 488.851,Z 657.404,A -85,B 0,C 180,E1 -6384.224,E2 -6384.224} C_VEL
LIN {X 0,Y 488.958,Z 657.389,A -85,B 0,C 180,E1 -6387.529,E2 -6387.529} C_VEL
LIN {X 0,Y 488.95,Z 657.393,A -85,B 0,C 180,E1 -6390.824,E2 -6390.824} C_VEL
LIN {X 0,Y 488.958,Z 657.389,A -85,B 0,C 180,E1 -6392.471,E2 -6392.471} C_VEL
LIN {X 0,Y 488.851,Z 657.404,A -85,B 0,C 180,E1 -6395.776,E2 -6395.776} C_VEL
LIN {X 0,Y 488.814,Z 657.407,A -85,B 0,C 180,E1 -6398.266,E2 -6398.266} C_VEL
LIN {X 0,Y 488.801,Z 657.413,A -85,B 0,C 180,E1 -6401.612,E2 -6401.612} C_VEL
LIN {X 0,Y 488.757,Z 657.416,A -85,B 0,C 180,E1 -6405,E2 -6405} C_VEL
LIN {X 0,Y 488.75,Z 657.416,A -85,B 0,C 180,E1 -6408.442,E2 -6408.442} C_VEL
LIN {X 0,Y 488.702,Z 657.42,A -85,B 0,C 180,E1 -6411.07,E2 -6411.07} C_VEL
LIN {X 0,Y 488.689,Z 657.426,A -85,B 0,C 180,E1 -6413.745,E2 -6413.745} C_VEL
LIN {X 0,Y 488.786,Z 657.41,A -85,B 0,C 180,E1 -6416.943,E2 -6416.943} C_VEL
LIN {X 0,Y 488.728,Z 657.422,A -85,B 0,C 180,E1 -6420.218,E2 -6420.218} C_VEL
LIN {X 0,Y 488.729,Z 657.417,A -85,B 0,C 180,E1 -6423.484,E2 -6423.484} C_VEL
LIN {X 0,Y 488.682,Z 657.428,A -85,B 0,C 180,E1 -6426.355,E2 -6426.355} C_VEL
LIN {X 0,Y 488.734,Z 657.416,A -85,B 0,C 180,E1 -6429.25,E2 -6429.25} C_VEL
LIN {X 0,Y 488.703,Z 657.419,A -85,B 0,C 180,E1 -6431.6,E2 -6431.6} C_VEL
LIN {X 0,Y 488.703,Z 657.426,A -85,B 0,C 180,E1 -6434.801,E2 -6434.801} C_VEL
LIN {X 0,Y 488.725,Z 657.418,A -85,B 0,C 180,E1 -6437.479,E2 -6437.479} C_VEL
LIN {X 0,Y 488.739,Z 657.419,A -85,B 0,C 180,E1 -6440.75,E2 -6440.75} C_VEL
LIN {X 0,Y 488.675,Z 657.403,A -85,B 0,C 180,E1 -6443.868,E2 -6443.868} C_VEL
LIN {X 0,Y 488.729,Z 657.417,A -85,B 0,C 180,E1 -6446.877,E2 -6446.877} C_VEL
LIN {X 0,Y 488.723,Z 657.403,A -85,B 0,C 180,E1 -6449.781,E2 -6449.781} C_VEL
LIN {X 0,Y 488.788,Z 657.396,A -85,B 0,C 180,E1 -6453.054,E2 -6453.054} C_VEL
LIN {X 0,Y 488.693,Z 657.419,A -85,B 0,C 180,E1 -6456.255,E2 -6456.255} C_VEL
LIN {X 0,Y 488.736,Z 657.413,A -85,B 0,C 180,E1 -6459.175,E2 -6459.175} C_VEL
LIN {X 0,Y 488.723,Z 657.412,A -85,B 0,C 180,E1 -6462.423,E2 -6462.423} C_VEL
LIN {X 0,Y 488.75,Z 657.411,A -85,B 0,C 180,E1 -6465,E2 -6465} C_VEL
LIN {X 0,Y 488.797,Z 657.41,A -85,B 0,C 180,E1 -6468.388,E2 -6468.388} C_VEL
LIN {X 0,Y 488.807,Z 657.402,A -85,B 0,C 180,E1 -6471.734,E2 -6471.734} C_VEL
LIN {X 0,Y 488.862,Z 657.401,A -85,B 0,C 180,E1 -6474.225,E2 -6474.225} C_VEL
LIN {X 0,Y 488.952,Z 657.378,A -85,B 0,C 180,E1 -6477.529,E2 -6477.529} C_VEL
LIN {X 0,Y 488.958,Z 657.387,A -85,B 0,C 180,E1 -6480,E2 -6480} C_VEL
LIN {X 0,Y 488.952,Z 657.386,A -85,B 0,C 180,E1 -6482.472,E2 -6482.472} C_VEL
LIN {X 0,Y 488.863,Z 657.397,A -85,B 0,C 180,E1 -6485.776,E2 -6485.776} C_VEL
LIN {X 0,Y 488.808,Z 657.395,A -85,B 0,C 180,E1 -6488.267,E2 -6488.267} C_VEL
LIN {X 0,Y 488.821,Z 657.401,A -85,B 0,C 180,E1 -6491.612,E2 -6491.612} C_VEL
LIN {X 0,Y 488.751,Z 657.414,A -85,B 0,C 180,E1 -6495.001,E2 -6495.001} C_VEL
LIN {X 0,Y 488.745,Z 657.408,A -85,B 0,C 180,E1 -6498.443,E2 -6498.443} C_VEL
LIN {X 0,Y 488.697,Z 657.422,A -85,B 0,C 180,E1 -6501.071,E2 -6501.071} C_VEL
LIN {X 0,Y 488.685,Z 657.426,A -85,B 0,C 180,E1 -6503.746,E2 -6503.746} C_VEL
LIN {X 0,Y 488.79,Z 657.401,A -85,B 0,C 180,E1 -6506.946,E2 -6506.946} C_VEL
LIN {X 0,Y 488.71,Z 657.412,A -85,B 0,C 180,E1 -6510.365,E2 -6510.365} C_VEL
LIN {X 0,Y 488.728,Z 657.418,A -85,B 0,C 180,E1 -6513.485,E2 -6513.485} C_VEL
LIN {X 0,Y 488.682,Z 657.413,A -85,B 0,C 180,E1 -6516.356,E2 -6516.356} C_VEL
LIN {X 0,Y 488.743,Z 657.413,A -85,B 0,C 180,E1 -6519.25,E2 -6519.25} C_VEL
LIN {X 0,Y 488.726,Z 657.404,A -85,B 0,C 180,E1 -6521.604,E2 -6521.604} C_VEL
LIN {X 0,Y 488.696,Z 657.424,A -85,B 0,C 180,E1 -6524.025,E2 -6524.025} C_VEL
LIN {X 0,Y 488.71,Z 657.421,A -85,B 0,C 180,E1 -6527.173,E2 -6527.173} C_VEL
LIN {X 0,Y 488.727,Z 657.415,A -85,B 0,C 180,E1 -6529.677,E2 -6529.677} C_VEL
LIN {X 0,Y 488.677,Z 657.394,A -85,B 0,C 180,E1 -6532.842,E2 -6532.842} C_VEL
LIN {X 0,Y 488.733,Z 657.496,A -85,B 0,C 180,E1 -6535.826,E2 -6535.826} C_VEL
LIN {X 0,Y 491.765,Z 669.513,A -85,B 0,C 180,E1 -6538.078,E2 -6538.078} C_VEL
LIN {X 0,Y 493.565,Z 676.998,A -85,B 0,C 180,E1 -6539.4,E2 -6539.4} C_VEL
LIN {X 0,Y 493.553,Z 682.586,A -85,B 0,C 180,E1 -6540.298,E2 -6540.298} C_VEL
LIN {X 0,Y 492.939,Z 694.243,A -85,B 0,C 180,E1 -6542.091,E2 -6542.091} C_VEL
LIN {X 0,Y 494.907,Z 702.344,A -85,B 0,C 180,E1 -6542.373,E2 -6542.373} C_VEL
LIN {X 0,Y 498.917,Z 719.013,A -85,B 0,C 180,E1 -6542.876,E2 -6542.876} C_VEL
LIN {X 0,Y 496.95,Z 896.191,A -85,B 0,C 180,E1 -6545.566,E2 -6545.566} C_VEL
LIN {X 0,Y 496.47,Z 909.327,A -85,B 0,C 180,E1 -6545.846,E2 -6545.846} C_VEL
LIN {X 0,Y 496.101,Z 921.693,A -85,B 0,C 180,E1 -6546.216,E2 -6546.216} C_VEL
LIN {X 0,Y 495.51,Z 934.82,A -85,B 0,C 180,E1 -6546.712,E2 -6546.712} C_VEL
LIN {X 0,Y 494.883,Z 947.306,A -85,B 0,C 180,E1 -6547.295,E2 -6547.295} C_VEL
LIN {X 0,Y 494.151,Z 960.133,A -85,B 0,C 180,E1 -6548.014,E2 -6548.014} C_VEL
LIN {X 0,Y 493.508,Z 970.762,A -85,B 0,C 180,E1 -6548.707,E2 -6548.707} C_VEL
LIN {X 0,Y 492.695,Z 983.205,A -85,B 0,C 180,E1 -6549.654,E2 -6549.654} C_VEL
LIN {X 0,Y 491.872,Z 994.88,A -85,B 0,C 180,E1 -6550.684,E2 -6550.684} C_VEL
LIN {X 0,Y 491.233,Z 1004.518,A -85,B 0,C 180,E1 -6551.655,E2 -6551.655} C_VEL
LIN {X 0,Y 490.59,Z 1013.793,A -85,B 0,C 180,E1 -6552.708,E2 -6552.708} C_VEL
LIN {X 0,Y 489.946,Z 1023.461,A -85,B 0,C 180,E1 -6553.961,E2 -6553.961} C_VEL
LIN {X 0,Y 489.444,Z 1032.056,A -85,B 0,C 180,E1 -6555.234,E2 -6555.234} C_VEL
LIN {X 0,Y 488.944,Z 1040.656,A -85,B 0,C 180,E1 -6556.704,E2 -6556.704} C_VEL
LIN {X 0,Y 488.675,Z 1047.686,A -85,B 0,C 180,E1 -6558.096,E2 -6558.096} C_VEL
LIN {X 0,Y 488.344,Z 1054.34,A -85,B 0,C 180,E1 -6559.637,E2 -6559.637} C_VEL
LIN {X 0,Y 488.18,Z 1058.984,A -85,B 0,C 180,E1 -6560.889,E2 -6560.889} C_VEL
LIN {X 0,Y 488.055,Z 1064.063,A -85,B 0,C 180,E1 -6562.554,E2 -6562.554} C_VEL
LIN {X 0,Y 488.008,Z 1066.667,A -85,B 0,C 180,E1 -6563.562,E2 -6563.562} C_VEL
LIN {X 0,Y 487.909,Z 1069.655,A -85,B 0,C 180,E1 -6565.042,E2 -6565.042} C_VEL
LIN {X 0,Y 487.945,Z 1072.081,A -85,B 0,C 180,E1 -6566.697,E2 -6566.697} C_VEL
LIN {X 0,Y 487.883,Z 1073.522,A -85,B 0,C 180,E1 -6568.349,E2 -6568.349} C_VEL
LIN {X 0,Y 487.814,Z 1074,A -85,B 0,C 180,E1 -6570,E2 -6570} C_VEL
LIN {X 0,Y 487.883,Z 1073.522,A -85,B 0,C 180,E1 -6571.651,E2 -6571.651} C_VEL
LIN {X 0,Y 487.945,Z 1072.081,A -85,B 0,C 180,E1 -6573.303,E2 -6573.303} C_VEL
LIN {X 0,Y 487.909,Z 1069.655,A -85,B 0,C 180,E1 -6574.958,E2 -6574.958} C_VEL
LIN {X 0,Y 488.028,Z 1066.21,A -85,B 0,C 180,E1 -6576.615,E2 -6576.615} C_VEL
LIN {X 0,Y 488.093,Z 1061.675,A -85,B 0,C 180,E1 -6578.279,E2 -6578.279} C_VEL
LIN {X 0,Y 488.23,Z 1055.958,A -85,B 0,C 180,E1 -6579.947,E2 -6579.947} C_VEL
LIN {X 0,Y 488.486,Z 1050.906,A -85,B 0,C 180,E1 -6581.199,E2 -6581.199} C_VEL
LIN {X 0,Y 488.822,Z 1042.878,A -85,B 0,C 180,E1 -6582.876,E2 -6582.876} C_VEL
LIN {X 0,Y 489.222,Z 1035.896,A -85,B 0,C 180,E1 -6584.135,E2 -6584.135} C_VEL
LIN {X 0,Y 489.734,Z 1027.929,A -85,B 0,C 180,E1 -6585.395,E2 -6585.395} C_VEL
LIN {X 0,Y 490.293,Z 1018.812,A -85,B 0,C 180,E1 -6586.659,E2 -6586.659} C_VEL
LIN {X 0,Y 490.811,Z 1010.239,A -85,B 0,C 180,E1 -6587.714,E2 -6587.714} C_VEL
LIN {X 0,Y 491.652,Z 998.367,A -85,B 0,C 180,E1 -6588.977,E2 -6588.977} C_VEL
LIN {X 0,Y 492.328,Z 988.094,A -85,B 0,C 180,E1 -6589.935,E2 -6589.935} C_VEL
LIN {X 0,Y 493.141,Z 976.519,A -85,B 0,C 180,E1 -6590.872,E2 -6590.872} C_VEL
LIN {X 0,Y 493.839,Z 964.483,A -85,B 0,C 180,E1 -6591.716,E2 -6591.716} C_VEL
LIN {X 0,Y 494.632,Z 952.307,A -85,B 0,C 180,E1 -6592.44,E2 -6592.44} C_VEL
LIN {X 0,Y 495.269,Z 939.006,A -85,B 0,C 180,E1 -6593.106,E2 -6593.106} C_VEL
LIN {X 0,Y 495.888,Z 926.171,A -85,B 0,C 180,E1 -6593.629,E2 -6593.629} C_VEL
LIN {X 0,Y 496.36,Z 913.246,A -85,B 0,C 180,E1 -6594.048,E2 -6594.048} C_VEL
LIN {X 0,Y 496.78,Z 900.409,A -85,B 0,C 180,E1 -6594.36,E2 -6594.36} C_VEL
LIN {X 0,Y 497.26,Z 874.373,A -85,B 0,C 180,E1 -6594.78,E2 -6594.78} C_VEL
LIN {X 0,Y 498.917,Z 718.852,A -85,B 0,C 180,E1 -6597.127,E2 -6597.127} C_VEL
LIN {X 0,Y 492.96,Z 694.293,A -85,B 0,C 180,E1 -6597.902,E2 -6597.902} C_VEL
LIN {X 0,Y 493.792,Z 678.474,A -85,B 0,C 180,E1 -6600.348,E2 -6600.348} C_VEL
LIN {X 0,Y 491.128,Z 666.811,A -85,B 0,C 180,E1 -6602.405,E2 -6602.405} C_VEL
LIN {X 0,Y 488.752,Z 657.52,A -85,B 0,C 180,E1 -6604.172,E2 -6604.172} C_VEL
LIN {X 0,Y 488.677,Z 657.394,A -85,B 0,C 180,E1 -6607.158,E2 -6607.158} C_VEL
LIN {X 0,Y 488.713,Z 657.417,A -85,B 0,C 180,E1 -6610.344,E2 -6610.344} C_VEL
LIN {X 0,Y 488.71,Z 657.421,A -85,B 0,C 180,E1 -6612.827,E2 -6612.827} C_VEL
LIN {X 0,Y 488.696,Z 657.424,A -85,B 0,C 180,E1 -6615.975,E2 -6615.975} C_VEL
LIN {X 0,Y 488.722,Z 657.404,A -85,B 0,C 180,E1 -6618.586,E2 -6618.586} C_VEL
LIN {X 0,Y 488.741,Z 657.414,A -85,B 0,C 180,E1 -6620.94,E2 -6620.94} C_VEL
LIN {X 0,Y 488.678,Z 657.411,A -85,B 0,C 180,E1 -6623.868,E2 -6623.868} C_VEL
LIN {X 0,Y 488.731,Z 657.415,A -85,B 0,C 180,E1 -6626.877,E2 -6626.877} C_VEL
LIN {X 0,Y 488.725,Z 657.406,A -85,B 0,C 180,E1 -6629.781,E2 -6629.781} C_VEL
LIN {X 0,Y 488.79,Z 657.401,A -85,B 0,C 180,E1 -6633.054,E2 -6633.054} C_VEL
LIN {X 0,Y 488.685,Z 657.426,A -85,B 0,C 180,E1 -6636.254,E2 -6636.254} C_VEL
LIN {X 0,Y 488.736,Z 657.415,A -85,B 0,C 180,E1 -6639.175,E2 -6639.175} C_VEL
LIN {X 0,Y 488.749,Z 657.407,A -85,B 0,C 180,E1 -6641.627,E2 -6641.627} C_VEL
LIN {X 0,Y 488.751,Z 657.415,A -85,B 0,C 180,E1 -6644.999,E2 -6644.999} C_VEL
LIN {X 0,Y 488.822,Z 657.401,A -85,B 0,C 180,E1 -6648.388,E2 -6648.388} C_VEL
LIN {X 0,Y 488.808,Z 657.396,A -85,B 0,C 180,E1 -6651.733,E2 -6651.733} C_VEL
LIN {X 0,Y 488.863,Z 657.397,A -85,B 0,C 180,E1 -6654.224,E2 -6654.224} C_VEL
LIN {X 0,Y 488.952,Z 657.386,A -85,B 0,C 180,E1 -6657.528,E2 -6657.528} C_VEL
LIN {X 0,Y 488.958,Z 657.387,A -85,B 0,C 180,E1 -6660,E2 -6660} C_VEL
LIN {X 0,Y 488.952,Z 657.377,A -85,B 0,C 180,E1 -6662.471,E2 -6662.471} C_VEL
LIN {X 0,Y 488.862,Z 657.402,A -85,B 0,C 180,E1 -6665.775,E2 -6665.775} C_VEL
LIN {X 0,Y 488.807,Z 657.403,A -85,B 0,C 180,E1 -6668.266,E2 -6668.266} C_VEL
LIN {X 0,Y 488.797,Z 657.411,A -85,B 0,C 180,E1 -6671.612,E2 -6671.612} C_VEL
LIN {X 0,Y 488.75,Z 657.411,A -85,B 0,C 180,E1 -6675,E2 -6675} C_VEL
LIN {X 0,Y 488.744,Z 657.416,A -85,B 0,C 180,E1 -6678.442,E2 -6678.442} C_VEL
LIN {X 0,Y 488.731,Z 657.412,A -85,B 0,C 180,E1 -6681.069,E2 -6681.069} C_VEL
LIN {X 0,Y 488.693,Z 657.419,A -85,B 0,C 180,E1 -6683.745,E2 -6683.745} C_VEL
LIN {X 0,Y 488.788,Z 657.396,A -85,B 0,C 180,E1 -6686.946,E2 -6686.946} C_VEL
LIN {X 0,Y 488.708,Z 657.407,A -85,B 0,C 180,E1 -6690.365,E2 -6690.365} C_VEL
LIN {X 0,Y 488.726,Z 657.414,A -85,B 0,C 180,E1 -6693.485,E2 -6693.485} C_VEL
LIN {X 0,Y 488.679,Z 657.403,A -85,B 0,C 180,E1 -6696.356,E2 -6696.356} C_VEL
LIN {X 0,Y 488.739,Z 657.419,A -85,B 0,C 180,E1 -6699.25,E2 -6699.25} C_VEL
LIN {X 0,Y 488.725,Z 657.418,A -85,B 0,C 180,E1 -6702.521,E2 -6702.521} C_VEL
LIN {X 0,Y 488.703,Z 657.426,A -85,B 0,C 180,E1 -6705.199,E2 -6705.199} C_VEL
LIN {X 0,Y 488.703,Z 657.419,A -85,B 0,C 180,E1 -6708.4,E2 -6708.4} C_VEL
LIN {X 0,Y 488.733,Z 657.418,A -85,B 0,C 180,E1 -6710.942,E2 -6710.942} C_VEL
LIN {X 0,Y 488.679,Z 657.426,A -85,B 0,C 180,E1 -6713.869,E2 -6713.869} C_VEL
LIN {X 0,Y 488.732,Z 657.417,A -85,B 0,C 180,E1 -6716.878,E2 -6716.878} C_VEL
LIN {X 0,Y 488.728,Z 657.422,A -85,B 0,C 180,E1 -6719.782,E2 -6719.782} C_VEL
LIN {X 0,Y 488.786,Z 657.41,A -85,B 0,C 180,E1 -6723.057,E2 -6723.057} C_VEL
LIN {X 0,Y 488.737,Z 657.418,A -85,B 0,C 180,E1 -6724.354,E2 -6724.354} C_VEL
LIN {X 0,Y 488.094,Z 657.501,A -85,B 0,C 180,E1 -6725.042,E2 -6725.042} C_VEL
LIN {X 0,Y 485.227,Z 657.861,A -85,B 0,C 180,E1 -6726.158,E2 -6726.158} C_VEL
LIN {X 0,Y 482.781,Z 658.164,A -85,B 0,C 180,E1 -6727.058,E2 -6727.058} C_VEL
LIN {X 0,Y 481.722,Z 658.294,A -85,B 0,C 180,E1 -6727.753,E2 -6727.753} C_VEL
LIN {X 0,Y 481.633,Z 658.303,A -85,B 0,C 180,E1 -6727.989,E2 -6727.989} C_VEL
LIN {X 0,Y 481.701,Z 658.296,A -85,B 0,C 180,E1 -6730.393,E2 -6730.393} C_VEL
LIN {X 0,Y 481.686,Z 658.294,A -85,B 0,C 180,E1 -6733.034,E2 -6733.034} C_VEL
LIN {X 0,Y 481.685,Z 658.296,A -85,B 0,C 180,E1 -6735.639,E2 -6735.639} C_VEL
LIN {X 0,Y 481.746,Z 658.291,A -85,B 0,C 180,E1 -6738.215,E2 -6738.215} C_VEL
LIN {X 0,Y 481.759,Z 658.286,A -85,B 0,C 180,E1 -6741.612,E2 -6741.612} C_VEL
LIN {X 0,Y 481.812,Z 658.28,A -85,B 0,C 180,E1 -6744.14,E2 -6744.14} C_VEL
LIN {X 0,Y 481.925,Z 658.266,A -85,B 0,C 180,E1 -6747.493,E2 -6747.493} C_VEL
LIN {X 0,Y 481.901,Z 658.271,A -85,B 0,C 180,E1 -6750.836,E2 -6750.836} C_VEL
LIN {X 0,Y 481.925,Z 658.266,A -85,B 0,C 180,E1 -6752.507,E2 -6752.507} C_VEL
LIN {X 0,Y 481.812,Z 658.28,A -85,B 0,C 180,E1 -6755.86,E2 -6755.86} C_VEL
LIN {X 0,Y 481.759,Z 658.286,A -85,B 0,C 180,E1 -6758.388,E2 -6758.388} C_VEL
LIN {X 0,Y 481.746,Z 658.291,A -85,B 0,C 180,E1 -6761.785,E2 -6761.785} C_VEL
LIN {X 0,Y 481.738,Z 658.291,A -85,B 0,C 180,E1 -6765.224,E2 -6765.224} C_VEL
LIN {X 0,Y 481.707,Z 658.292,A -85,B 0,C 180,E1 -6768.721,E2 -6768.721} C_VEL
LIN {X 0,Y 481.642,Z 658.302,A -85,B 0,C 180,E1 -6771.394,E2 -6771.394} C_VEL
LIN {X 0,Y 481.672,Z 658.301,A -85,B 0,C 180,E1 -6774.113,E2 -6774.113} C_VEL
LIN {X 0,Y 481.741,Z 658.287,A -85,B 0,C 180,E1 -6777.139,E2 -6777.139} C_VEL
LIN {X 0,Y 481.682,Z 658.298,A -85,B 0,C 180,E1 -6779.74,E2 -6779.74} C_VEL
LIN {X 0,Y 481.667,Z 658.3,A -85,B 0,C 180,E1 -6782.674,E2 -6782.674} C_VEL
LIN {X 0,Y 481.636,Z 658.3,A -85,B 0,C 180,E1 -6785.708,E2 -6785.708} C_VEL
LIN {X 0,Y 481.706,Z 658.291,A -85,B 0,C 180,E1 -6789.353,E2 -6789.353} C_VEL
LIN {X 0,Y 481.64,Z 658.301,A -85,B 0,C 180,E1 -6792.16,E2 -6792.16} C_VEL
LIN {X 0,Y 481.651,Z 658.299,A -85,B 0,C 180,E1 -6795.542,E2 -6795.542} C_VEL
LIN {X 0,Y 481.667,Z 658.296,A -85,B 0,C 180,E1 -6798.084,E2 -6798.084} C_VEL
LIN {X 0,Y 481.694,Z 658.295,A -85,B 0,C 180,E1 -6801.144,E2 -6801.144} C_VEL
LIN {X 0,Y 481.658,Z 658.28,A -85,B 0,C 180,E1 -6804.794,E2 -6804.794} C_VEL
LIN {X 0,Y 481.663,Z 658.304,A -85,B 0,C 180,E1 -6807.326,E2 -6807.326} C_VEL
LIN {X 0,Y 481.677,Z 658.276,A -85,B 0,C 180,E1 -6810.259,E2 -6810.259} C_VEL
LIN {X 0,Y 481.742,Z 658.274,A -85,B 0,C 180,E1 -6813.112,E2 -6813.112} C_VEL
LIN {X 0,Y 481.673,Z 658.297,A -85,B 0,C 180,E1 -6815.887,E2 -6815.887} C_VEL
LIN {X 0,Y 481.7,Z 658.289,A -85,B 0,C 180,E1 -6819.025,E2 -6819.025} C_VEL
LIN {X 0,Y 481.696,Z 658.288,A -85,B 0,C 180,E1 -6822.158,E2 -6822.158} C_VEL
LIN {X 0,Y 481.731,Z 658.286,A -85,B 0,C 180,E1 -6824.776,E2 -6824.776} C_VEL
LIN {X 0,Y 481.741,Z 658.285,A -85,B 0,C 180,E1 -6828.215,E2 -6828.215} C_VEL
LIN {X 0,Y 481.753,Z 658.28,A -85,B 0,C 180,E1 -6831.612,E2 -6831.612} C_VEL
LIN {X 0,Y 481.821,Z 658.277,A -85,B 0,C 180,E1 -6834.14,E2 -6834.14} C_VEL
LIN {X 0,Y 481.919,Z 658.254,A -85,B 0,C 180,E1 -6837.493,E2 -6837.493} C_VEL
LIN {X 0,Y 481.929,Z 658.263,A -85,B 0,C 180,E1 -6840,E2 -6840} C_VEL
LIN {X 0,Y 481.919,Z 658.262,A -85,B 0,C 180,E1 -6842.508,E2 -6842.508} C_VEL
LIN {X 0,Y 481.821,Z 658.274,A -85,B 0,C 180,E1 -6845.861,E2 -6845.861} C_VEL
LIN {X 0,Y 481.754,Z 658.274,A -85,B 0,C 180,E1 -6848.389,E2 -6848.389} C_VEL
LIN {X 0,Y 481.786,Z 658.275,A -85,B 0,C 180,E1 -6851.784,E2 -6851.784} C_VEL
LIN {X 0,Y 481.732,Z 658.292,A -85,B 0,C 180,E1 -6855.225,E2 -6855.225} C_VEL
LIN {X 0,Y 481.702,Z 658.286,A -85,B 0,C 180,E1 -6858.722,E2 -6858.722} C_VEL
LIN {X 0,Y 481.637,Z 658.302,A -85,B 0,C 180,E1 -6861.395,E2 -6861.395} C_VEL
LIN {X 0,Y 481.668,Z 658.297,A -85,B 0,C 180,E1 -6864.114,E2 -6864.114} C_VEL
LIN {X 0,Y 481.743,Z 658.28,A -85,B 0,C 180,E1 -6867.141,E2 -6867.141} C_VEL
LIN {X 0,Y 481.679,Z 658.272,A -85,B 0,C 180,E1 -6869.741,E2 -6869.741} C_VEL
LIN {X 0,Y 481.665,Z 658.296,A -85,B 0,C 180,E1 -6872.675,E2 -6872.675} C_VEL
LIN {X 0,Y 481.635,Z 658.286,A -85,B 0,C 180,E1 -6875.71,E2 -6875.71} C_VEL
LIN {X 0,Y 481.716,Z 658.289,A -85,B 0,C 180,E1 -6879.356,E2 -6879.356} C_VEL
LIN {X 0,Y 481.669,Z 658.289,A -85,B 0,C 180,E1 -6882.158,E2 -6882.158} C_VEL
LIN {X 0,Y 481.654,Z 658.295,A -85,B 0,C 180,E1 -6884.458,E2 -6884.458} C_VEL
LIN {X 0,Y 481.648,Z 658.3,A -85,B 0,C 180,E1 -6887.841,E2 -6887.841} C_VEL
LIN {X 0,Y 481.675,Z 658.303,A -85,B 0,C 180,E1 -6890.652,E2 -6890.652} C_VEL
LIN {X 0,Y 481.626,Z 658.267,A -85,B 0,C 180,E1 -6893.376,E2 -6893.376} C_VEL
LIN {X 0,Y 481.721,Z 658.5,A -85,B 0,C 180,E1 -6895.494,E2 -6895.494} C_VEL
LIN {X 0,Y 484.864,Z 670.776,A -85,B 0,C 180,E1 -6897.814,E2 -6897.814} C_VEL
LIN {X 0,Y 486.898,Z 679.681,A -85,B 0,C 180,E1 -6899.417,E2 -6899.417} C_VEL
LIN {X 0,Y 486.214,Z 694.068,A -85,B 0,C 180,E1 -6901.677,E2 -6901.677} C_VEL
LIN {X 0,Y 492.571,Z 720.249,A -85,B 0,C 180,E1 -6902.52,E2 -6902.52} C_VEL
LIN {X 0,Y 490.673,Z 884.912,A -85,B 0,C 180,E1 -6905.034,E2 -6905.034} C_VEL
LIN {X 0,Y 490.175,Z 906.185,A -85,B 0,C 180,E1 -6905.431,E2 -6905.431} C_VEL
LIN {X 0,Y 489.552,Z 920.738,A -85,B 0,C 180,E1 -6905.85,E2 -6905.85} C_VEL
LIN {X 0,Y 488.983,Z 934.611,A -85,B 0,C 180,E1 -6906.383,E2 -6906.383} C_VEL
LIN {X 0,Y 488.353,Z 946.003,A -85,B 0,C 180,E1 -6906.912,E2 -6906.912} C_VEL
LIN {X 0,Y 487.613,Z 958.894,A -85,B 0,C 180,E1 -6907.634,E2 -6907.634} C_VEL
LIN {X 0,Y 486.788,Z 970.553,A -85,B 0,C 180,E1 -6908.399,E2 -6908.399} C_VEL
LIN {X 0,Y 485.96,Z 982.997,A -85,B 0,C 180,E1 -6909.359,E2 -6909.359} C_VEL
LIN {X 0,Y 485.15,Z 993.846,A -85,B 0,C 180,E1 -6910.323,E2 -6910.323} C_VEL
LIN {X 0,Y 484.386,Z 1004.309,A -85,B 0,C 180,E1 -6911.386,E2 -6911.386} C_VEL
LIN {X 0,Y 483.715,Z 1013.584,A -85,B 0,C 180,E1 -6912.454,E2 -6912.454} C_VEL
LIN {X 0,Y 482.969,Z 1023.928,A -85,B 0,C 180,E1 -6913.823,E2 -6913.823} C_VEL
LIN {X 0,Y 482.503,Z 1031.849,A -85,B 0,C 180,E1 -6915.017,E2 -6915.017} C_VEL
LIN {X 0,Y 481.945,Z 1040.448,A -85,B 0,C 180,E1 -6916.508,E2 -6916.508} C_VEL
LIN {X 0,Y 481.63,Z 1047.251,A -85,B 0,C 180,E1 -6917.868,E2 -6917.868} C_VEL
LIN {X 0,Y 481.283,Z 1054.132,A -85,B 0,C 180,E1 -6919.483,E2 -6919.483} C_VEL
LIN {X 0,Y 481.107,Z 1058.777,A -85,B 0,C 180,E1 -6920.753,E2 -6920.753} C_VEL
LIN {X 0,Y 480.978,Z 1063.864,A -85,B 0,C 180,E1 -6922.444,E2 -6922.444} C_VEL
LIN {X 0,Y 480.918,Z 1066.758,A -85,B 0,C 180,E1 -6923.58,E2 -6923.58} C_VEL
LIN {X 0,Y 480.835,Z 1069.516,A -85,B 0,C 180,E1 -6924.969,E2 -6924.969} C_VEL
LIN {X 0,Y 480.85,Z 1071.974,A -85,B 0,C 180,E1 -6926.648,E2 -6926.648} C_VEL
LIN {X 0,Y 480.784,Z 1073.432,A -85,B 0,C 180,E1 -6928.325,E2 -6928.325} C_VEL
LIN {X 0,Y 480.738,Z 1073.914,A -85,B 0,C 180,E1 -6930,E2 -6930} C_VEL
LIN {X 0,Y 480.784,Z 1073.432,A -85,B 0,C 180,E1 -6931.675,E2 -6931.675} C_VEL
LIN {X 0,Y 480.85,Z 1071.974,A -85,B 0,C 180,E1 -6933.352,E2 -6933.352} C_VEL
LIN {X 0,Y 480.835,Z 1069.516,A -85,B 0,C 180,E1 -6935.031,E2 -6935.031} C_VEL
LIN {X 0,Y 480.951,Z 1066.034,A -85,B 0,C 180,E1 -6936.713,E2 -6936.713} C_VEL
LIN {X 0,Y 481.021,Z 1061.468,A -85,B 0,C 180,E1 -6938.401,E2 -6938.401} C_VEL
LIN {X 0,Y 481.184,Z 1055.751,A -85,B 0,C 180,E1 -6940.094,E2 -6940.094} C_VEL
LIN {X 0,Y 481.439,Z 1050.698,A -85,B 0,C 180,E1 -6941.365,E2 -6941.365} C_VEL
LIN {X 0,Y 481.828,Z 1042.67,A -85,B 0,C 180,E1 -6943.066,E2 -6943.066} C_VEL
LIN {X 0,Y 482.218,Z 1035.687,A -85,B 0,C 180,E1 -6944.345,E2 -6944.345} C_VEL
LIN {X 0,Y 482.779,Z 1027.72,A -85,B 0,C 180,E1 -6945.623,E2 -6945.623} C_VEL
LIN {X 0,Y 483.37,Z 1018.603,A -85,B 0,C 180,E1 -6946.905,E2 -6946.905} C_VEL
LIN {X 0,Y 483.948,Z 1010.03,A -85,B 0,C 180,E1 -6947.974,E2 -6947.974} C_VEL
LIN {X 0,Y 484.766,Z 999.248,A -85,B 0,C 180,E1 -6949.148,E2 -6949.148} C_VEL
LIN {X 0,Y 485.551,Z 988.015,A -85,B 0,C 180,E1 -6950.214,E2 -6950.214} C_VEL
LIN {X 0,Y 486.439,Z 976.311,A -85,B 0,C 180,E1 -6951.173,E2 -6951.173} C_VEL
LIN {X 0,Y 487.185,Z 964.276,A -85,B 0,C 180,E1 -6952.028,E2 -6952.028} C_VEL
LIN {X 0,Y 488.021,Z 951.811,A -85,B 0,C 180,E1 -6952.777,E2 -6952.777} C_VEL
LIN {X 0,Y 488.68,Z 939.398,A -85,B 0,C 180,E1 -6953.408,E2 -6953.408} C_VEL
LIN {X 0,Y 489.37,Z 925.965,A -85,B 0,C 180,E1 -6953.963,E2 -6953.963} C_VEL
LIN {X 0,Y 489.879,Z 913.041,A -85,B 0,C 180,E1 -6954.387,E2 -6954.387} C_VEL
LIN {X 0,Y 490.329,Z 900.203,A -85,B 0,C 180,E1 -6954.702,E2 -6954.702} C_VEL
LIN {X 0,Y 490.818,Z 874.167,A -85,B 0,C 180,E1 -6955.128,E2 -6955.128} C_VEL
LIN {X 0,Y 492.577,Z 720.151,A -85,B 0,C 180,E1 -6957.481,E2 -6957.481} C_VEL
LIN {X 0,Y 486.243,Z 694.117,A -85,B 0,C 180,E1 -6958.316,E2 -6958.316} C_VEL
LIN {X 0,Y 486.974,Z 681.151,A -85,B 0,C 180,E1 -6960.338,E2 -6960.338} C_VEL
LIN {X 0,Y 486.37,Z 677.123,A -85,B 0,C 180,E1 -6961.037,E2 -6961.037} C_VEL
LIN {X 0,Y 482.952,Z 663.307,A -85,B 0,C 180,E1 -6963.571,E2 -6963.571} C_VEL
LIN {X 0,Y 481.707,Z 658.365,A -85,B 0,C 180,E1 -6964.564,E2 -6964.564} C_VEL
LIN {X 0,Y 481.651,Z 658.283,A -85,B 0,C 180,E1 -6968.007,E2 -6968.007} C_VEL
LIN {X 0,Y 481.657,Z 658.292,A -85,B 0,C 180,E1 -6971.04,E2 -6971.04} C_VEL
LIN {X 0,Y 481.653,Z 658.285,A -85,B 0,C 180,E1 -6974.359,E2 -6974.359} C_VEL
LIN {X 0,Y 481.683,Z 658.295,A -85,B 0,C 180,E1 -6976.845,E2 -6976.845} C_VEL
LIN {X 0,Y 481.706,Z 658.291,A -85,B 0,C 180,E1 -6980.063,E2 -6980.063} C_VEL
LIN {X 0,Y 481.625,Z 658.294,A -85,B 0,C 180,E1 -6983.375,E2 -6983.375} C_VEL
LIN {X 0,Y 481.701,Z 658.295,A -85,B 0,C 180,E1 -6986.329,E2 -6986.329} C_VEL
LIN {X 0,Y 481.65,Z 658.292,A -85,B 0,C 180,E1 -6989.415,E2 -6989.415} C_VEL
LIN {X 0,Y 481.694,Z 658.271,A -85,B 0,C 180,E1 -6992.168,E2 -6992.168} C_VEL
LIN {X 0,Y 481.709,Z 658.291,A -85,B 0,C 180,E1 -6994.969,E2 -6994.969} C_VEL
LIN {X 0,Y 481.643,Z 658.291,A -85,B 0,C 180,E1 -6997.704,E2 -6997.704} C_VEL
LIN {X 0,Y 481.698,Z 658.298,A -85,B 0,C 180,E1 -7000.393,E2 -7000.393} C_VEL
LIN {X 0,Y 481.682,Z 658.296,A -85,B 0,C 180,E1 -7003.034,E2 -7003.034} C_VEL
LIN {X 0,Y 481.681,Z 658.291,A -85,B 0,C 180,E1 -7005.638,E2 -7005.638} C_VEL
LIN {X 0,Y 481.786,Z 658.276,A -85,B 0,C 180,E1 -7008.216,E2 -7008.216} C_VEL
LIN {X 0,Y 481.754,Z 658.275,A -85,B 0,C 180,E1 -7011.611,E2 -7011.611} C_VEL
LIN {X 0,Y 481.821,Z 658.274,A -85,B 0,C 180,E1 -7014.139,E2 -7014.139} C_VEL
LIN {X 0,Y 481.919,Z 658.261,A -85,B 0,C 180,E1 -7017.492,E2 -7017.492} C_VEL
LIN {X 0,Y 481.929,Z 658.262,A -85,B 0,C 180,E1 -7020,E2 -7020} C_VEL
LIN {X 0,Y 481.919,Z 658.253,A -85,B 0,C 180,E1 -7022.507,E2 -7022.507} C_VEL
LIN {X 0,Y 481.821,Z 658.278,A -85,B 0,C 180,E1 -7025.86,E2 -7025.86} C_VEL
LIN {X 0,Y 481.753,Z 658.281,A -85,B 0,C 180,E1 -7028.388,E2 -7028.388} C_VEL
LIN {X 0,Y 481.741,Z 658.286,A -85,B 0,C 180,E1 -7031.785,E2 -7031.785} C_VEL
LIN {X 0,Y 481.731,Z 658.286,A -85,B 0,C 180,E1 -7035.224,E2 -7035.224} C_VEL
LIN {X 0,Y 481.701,Z 658.29,A -85,B 0,C 180,E1 -7038.722,E2 -7038.722} C_VEL
LIN {X 0,Y 481.666,Z 658.293,A -85,B 0,C 180,E1 -7041.393,E2 -7041.393} C_VEL
LIN {X 0,Y 481.673,Z 658.297,A -85,B 0,C 180,E1 -7044.113,E2 -7044.113} C_VEL
LIN {X 0,Y 481.741,Z 658.272,A -85,B 0,C 180,E1 -7047.141,E2 -7047.141} C_VEL
LIN {X 0,Y 481.677,Z 658.276,A -85,B 0,C 180,E1 -7049.741,E2 -7049.741} C_VEL
LIN {X 0,Y 481.663,Z 658.304,A -85,B 0,C 180,E1 -7052.674,E2 -7052.674} C_VEL
LIN {X 0,Y 481.633,Z 658.279,A -85,B 0,C 180,E1 -7055.709,E2 -7055.709} C_VEL
LIN {X 0,Y 481.71,Z 658.294,A -85,B 0,C 180,E1 -7059.355,E2 -7059.355} C_VEL
LIN {X 0,Y 481.667,Z 658.296,A -85,B 0,C 180,E1 -7062.158,E2 -7062.158} C_VEL
LIN {X 0,Y 481.651,Z 658.299,A -85,B 0,C 180,E1 -7064.458,E2 -7064.458} C_VEL
LIN {X 0,Y 481.64,Z 658.301,A -85,B 0,C 180,E1 -7067.84,E2 -7067.84} C_VEL
LIN {X 0,Y 481.706,Z 658.291,A -85,B 0,C 180,E1 -7070.647,E2 -7070.647} C_VEL
LIN {X 0,Y 481.636,Z 658.3,A -85,B 0,C 180,E1 -7074.292,E2 -7074.292} C_VEL
LIN {X 0,Y 481.667,Z 658.3,A -85,B 0,C 180,E1 -7077.326,E2 -7077.326} C_VEL
LIN {X 0,Y 481.681,Z 658.298,A -85,B 0,C 180,E1 -7080.26,E2 -7080.26} C_VEL
LIN {X 0,Y 481.74,Z 658.288,A -85,B 0,C 180,E1 -7083.113,E2 -7083.113} C_VEL
LIN {X 0,Y 481.672,Z 658.301,A -85,B 0,C 180,E1 -7085.887,E2 -7085.887} C_VEL
LIN {X 0,Y 481.633,Z 658.303,A -85,B 0,C 180,E1 -7087.989,E2 -7087.989} C_VEL
LIN {X 0,Y 480.965,Z 658.387,A -85,B 0,C 180,E1 -7088.687,E2 -7088.687} C_VEL
LIN {X 0,Y 478.136,Z 658.739,A -85,B 0,C 180,E1 -7089.821,E2 -7089.821} C_VEL
LIN {X 0,Y 475.752,Z 659.036,A -85,B 0,C 180,E1 -7090.735,E2 -7090.735} C_VEL
LIN {X 0,Y 474.732,Z 659.162,A -85,B 0,C 180,E1 -7091.441,E2 -7091.441} C_VEL
LIN {X 0,Y 474.65,Z 659.173,A -85,B 0,C 180,E1 -7091.68,E2 -7091.68} C_VEL
LIN {X 0,Y 474.695,Z 659.169,A -85,B 0,C 180,E1 -7094.545,E2 -7094.545} C_VEL
LIN {X 0,Y 474.7,Z 659.167,A -85,B 0,C 180,E1 -7098.038,E2 -7098.038} C_VEL
LIN {X 0,Y 474.724,Z 659.162,A -85,B 0,C 180,E1 -7101.487,E2 -7101.487} C_VEL
LIN {X 0,Y 474.775,Z 659.157,A -85,B 0,C 180,E1 -7104.053,E2 -7104.053} C_VEL
LIN {X 0,Y 474.891,Z 659.143,A -85,B 0,C 180,E1 -7107.455,E2 -7107.455} C_VEL
LIN {X 0,Y 474.908,Z 659.14,A -85,B 0,C 180,E1 -7110,E2 -7110} C_VEL
LIN {X 0,Y 474.891,Z 659.143,A -85,B 0,C 180,E1 -7112.545,E2 -7112.545} C_VEL
LIN {X 0,Y 474.775,Z 659.157,A -85,B 0,C 180,E1 -7115.947,E2 -7115.947} C_VEL
LIN {X 0,Y 474.724,Z 659.162,A -85,B 0,C 180,E1 -7118.513,E2 -7118.513} C_VEL
LIN {X 0,Y 474.7,Z 659.167,A -85,B 0,C 180,E1 -7121.962,E2 -7121.962} C_VEL
LIN {X 0,Y 474.695,Z 659.169,A -85,B 0,C 180,E1 -7125.455,E2 -7125.455} C_VEL
LIN {X 0,Y 474.66,Z 659.171,A -85,B 0,C 180,E1 -7129.01,E2 -7129.01} C_VEL
LIN {X 0,Y 474.586,Z 659.184,A -85,B 0,C 180,E1 -7131.728,E2 -7131.728} C_VEL
LIN {X 0,Y 474.654,Z 659.172,A -85,B 0,C 180,E1 -7134.492,E2 -7134.492} C_VEL
LIN {X 0,Y 474.693,Z 659.166,A -85,B 0,C 180,E1 -7137.338,E2 -7137.338} C_VEL
LIN {X 0,Y 474.604,Z 659.178,A -85,B 0,C 180,E1 -7140.811,E2 -7140.811} C_VEL
LIN {X 0,Y 474.631,Z 659.177,A -85,B 0,C 180,E1 -7143.984,E2 -7143.984} C_VEL
LIN {X 0,Y 474.568,Z 659.184,A -85,B 0,C 180,E1 -7146.9,E2 -7146.9} C_VEL
LIN {X 0,Y 474.642,Z 659.171,A -85,B 0,C 180,E1 -7149.65,E2 -7149.65} C_VEL
LIN {X 0,Y 474.606,Z 659.182,A -85,B 0,C 180,E1 -7152.934,E2 -7152.934} C_VEL
LIN {X 0,Y 474.61,Z 659.175,A -85,B 0,C 180,E1 -7155.896,E2 -7155.896} C_VEL
LIN {X 0,Y 474.638,Z 659.178,A -85,B 0,C 180,E1 -7159.038,E2 -7159.038} C_VEL
LIN {X 0,Y 474.61,Z 659.171,A -85,B 0,C 180,E1 -7161.702,E2 -7161.702} C_VEL
LIN {X 0,Y 474.62,Z 659.155,A -85,B 0,C 180,E1 -7164.726,E2 -7164.726} C_VEL
LIN {X 0,Y 474.627,Z 659.174,A -85,B 0,C 180,E1 -7167.788,E2 -7167.788} C_VEL
LIN {X 0,Y 474.621,Z 659.15,A -85,B 0,C 180,E1 -7170.883,E2 -7170.883} C_VEL
LIN {X 0,Y 474.656,Z 659.164,A -85,B 0,C 180,E1 -7173.629,E2 -7173.629} C_VEL
LIN {X 0,Y 474.631,Z 659.169,A -85,B 0,C 180,E1 -7176.639,E2 -7176.639} C_VEL
LIN {X 0,Y 474.665,Z 659.166,A -85,B 0,C 180,E1 -7179.186,E2 -7179.186} C_VEL
LIN {X 0,Y 474.646,Z 659.168,A -85,B 0,C 180,E1 -7181.884,E2 -7181.884} C_VEL
LIN {X 0,Y 474.688,Z 659.165,A -85,B 0,C 180,E1 -7184.544,E2 -7184.544} C_VEL
LIN {X 0,Y 474.694,Z 659.159,A -85,B 0,C 180,E1 -7188.038,E2 -7188.038} C_VEL
LIN {X 0,Y 474.718,Z 659.155,A -85,B 0,C 180,E1 -7191.487,E2 -7191.487} C_VEL
LIN {X 0,Y 474.781,Z 659.152,A -85,B 0,C 180,E1 -7194.053,E2 -7194.053} C_VEL
LIN {X 0,Y 474.885,Z 659.129,A -85,B 0,C 180,E1 -7197.456,E2 -7197.456} C_VEL
LIN {X 0,Y 474.867,Z 659.145,A -85,B 0,C 180,E1 -7200.848,E2 -7200.848} C_VEL
LIN {X 0,Y 474.885,Z 659.137,A -85,B 0,C 180,E1 -7202.545,E2 -7202.545} C_VEL
LIN {X 0,Y 474.781,Z 659.151,A -85,B 0,C 180,E1 -7205.948,E2 -7205.948} C_VEL
LIN {X 0,Y 474.719,Z 659.151,A -85,B 0,C 180,E1 -7208.514,E2 -7208.514} C_VEL
LIN {X 0,Y 474.73,Z 659.153,A -85,B 0,C 180,E1 -7211.962,E2 -7211.962} C_VEL
LIN {X 0,Y 474.67,Z 659.167,A -85,B 0,C 180,E1 -7215.768,E2 -7215.768} C_VEL
LIN {X 0,Y 474.656,Z 659.166,A -85,B 0,C 180,E1 -7219.011,E2 -7219.011} C_VEL
LIN {X 0,Y 474.581,Z 659.175,A -85,B 0,C 180,E1 -7221.729,E2 -7221.729} C_VEL
LIN {X 0,Y 474.65,Z 659.169,A -85,B 0,C 180,E1 -7224.493,E2 -7224.493} C_VEL
LIN {X 0,Y 474.69,Z 659.152,A -85,B 0,C 180,E1 -7227.339,E2 -7227.339} C_VEL
LIN {X 0,Y 474.602,Z 659.169,A -85,B 0,C 180,E1 -7230.812,E2 -7230.812} C_VEL
LIN {X 0,Y 474.63,Z 659.17,A -85,B 0,C 180,E1 -7233.985,E2 -7233.985} C_VEL
LIN {X 0,Y 474.569,Z 659.175,A -85,B 0,C 180,E1 -7236.901,E2 -7236.901} C_VEL
LIN {X 0,Y 474.66,Z 659.17,A -85,B 0,C 180,E1 -7239.654,E2 -7239.654} C_VEL
LIN {X 0,Y 474.646,Z 659.173,A -85,B 0,C 180,E1 -7242.931,E2 -7242.931} C_VEL
LIN {X 0,Y 474.609,Z 659.164,A -85,B 0,C 180,E1 -7245.897,E2 -7245.897} C_VEL
LIN {X 0,Y 474.627,Z 659.167,A -85,B 0,C 180,E1 -7249.041,E2 -7249.041} C_VEL
LIN {X 0,Y 474.605,Z 659.167,A -85,B 0,C 180,E1 -7251.705,E2 -7251.705} C_VEL
LIN {X 0,Y 474.657,Z 659.253,A -85,B 0,C 180,E1 -7255.054,E2 -7255.054} C_VEL
LIN {X 0,Y 477.542,Z 670.553,A -85,B 0,C 180,E1 -7257.267,E2 -7257.267} C_VEL
LIN {X 0,Y 480.012,Z 680.888,A -85,B 0,C 180,E1 -7259.174,E2 -7259.174} C_VEL
LIN {X 0,Y 479.92,Z 686.755,A -85,B 0,C 180,E1 -7260.14,E2 -7260.14} C_VEL
LIN {X 0,Y 479.527,Z 693.979,A -85,B 0,C 180,E1 -7261.257,E2 -7261.257} C_VEL
LIN {X 0,Y 486.264,Z 721.503,A -85,B 0,C 180,E1 -7262.157,E2 -7262.157} C_VEL
LIN {X 0,Y 484.235,Z 885.109,A -85,B 0,C 180,E1 -7264.686,E2 -7264.686} C_VEL
LIN {X 0,Y 483.706,Z 905.979,A -85,B 0,C 180,E1 -7265.081,E2 -7265.081} C_VEL
LIN {X 0,Y 483.068,Z 920.532,A -85,B 0,C 180,E1 -7265.504,E2 -7265.504} C_VEL
LIN {X 0,Y 482.449,Z 934.405,A -85,B 0,C 180,E1 -7266.043,E2 -7266.043} C_VEL
LIN {X 0,Y 481.802,Z 945.797,A -85,B 0,C 180,E1 -7266.579,E2 -7266.579} C_VEL
LIN {X 0,Y 480.945,Z 959.146,A -85,B 0,C 180,E1 -7267.338,E2 -7267.338} C_VEL
LIN {X 0,Y 480.132,Z 970.345,A -85,B 0,C 180,E1 -7268.084,E2 -7268.084} C_VEL
LIN {X 0,Y 479.258,Z 982.79,A -85,B 0,C 180,E1 -7269.057,E2 -7269.057} C_VEL
LIN {X 0,Y 478.31,Z 994.468,A -85,B 0,C 180,E1 -7270.115,E2 -7270.115} C_VEL
LIN {X 0,Y 477.555,Z 1004.1,A -85,B 0,C 180,E1 -7271.11,E2 -7271.11} C_VEL
LIN {X 0,Y 476.824,Z 1013.375,A -85,B 0,C 180,E1 -7272.192,E2 -7272.192} C_VEL
LIN {X 0,Y 476.122,Z 1023.261,A -85,B 0,C 180,E1 -7273.515,E2 -7273.515} C_VEL
LIN {X 0,Y 475.556,Z 1031.64,A -85,B 0,C 180,E1 -7274.793,E2 -7274.793} C_VEL
LIN {X 0,Y 474.927,Z 1040.239,A -85,B 0,C 180,E1 -7276.304,E2 -7276.304} C_VEL
LIN {X 0,Y 474.589,Z 1047.485,A -85,B 0,C 180,E1 -7277.786,E2 -7277.786} C_VEL
LIN {X 0,Y 474.226,Z 1053.924,A -85,B 0,C 180,E1 -7279.325,E2 -7279.325} C_VEL
LIN {X 0,Y 474.015,Z 1058.569,A -85,B 0,C 180,E1 -7280.614,E2 -7280.614} C_VEL
LIN {X 0,Y 473.898,Z 1063.657,A -85,B 0,C 180,E1 -7282.33,E2 -7282.33} C_VEL
LIN {X 0,Y 473.786,Z 1067.643,A -85,B 0,C 180,E1 -7284.04,E2 -7284.04} C_VEL
LIN {X 0,Y 473.763,Z 1069.311,A -85,B 0,C 180,E1 -7284.894,E2 -7284.894} C_VEL
LIN {X 0,Y 473.743,Z 1071.768,A -85,B 0,C 180,E1 -7286.598,E2 -7286.598} C_VEL
LIN {X 0,Y 473.689,Z 1073.226,A -85,B 0,C 180,E1 -7288.3,E2 -7288.3} C_VEL
LIN {X 0,Y 473.665,Z 1073.71,A -85,B 0,C 180,E1 -7290,E2 -7290} C_VEL
LIN {X 0,Y 473.689,Z 1073.226,A -85,B 0,C 180,E1 -7291.7,E2 -7291.7} C_VEL
LIN {X 0,Y 473.743,Z 1071.768,A -85,B 0,C 180,E1 -7293.402,E2 -7293.402} C_VEL
LIN {X 0,Y 473.763,Z 1069.311,A -85,B 0,C 180,E1 -7295.106,E2 -7295.106} C_VEL
LIN {X 0,Y 473.866,Z 1065.828,A -85,B 0,C 180,E1 -7296.814,E2 -7296.814} C_VEL
LIN {X 0,Y 473.935,Z 1061.261,A -85,B 0,C 180,E1 -7298.528,E2 -7298.528} C_VEL
LIN {X 0,Y 474.14,Z 1055.544,A -85,B 0,C 180,E1 -7300.246,E2 -7300.246} C_VEL
LIN {X 0,Y 474.401,Z 1050.49,A -85,B 0,C 180,E1 -7301.536,E2 -7301.536} C_VEL
LIN {X 0,Y 474.812,Z 1042.462,A -85,B 0,C 180,E1 -7303.263,E2 -7303.263} C_VEL
LIN {X 0,Y 475.226,Z 1035.478,A -85,B 0,C 180,E1 -7304.56,E2 -7304.56} C_VEL
LIN {X 0,Y 475.822,Z 1027.622,A -85,B 0,C 180,E1 -7305.841,E2 -7305.841} C_VEL
LIN {X 0,Y 476.47,Z 1018.394,A -85,B 0,C 180,E1 -7307.157,E2 -7307.157} C_VEL
LIN {X 0,Y 477.108,Z 1009.822,A -85,B 0,C 180,E1 -7308.241,E2 -7308.241} C_VEL
LIN {X 0,Y 477.973,Z 999.039,A -85,B 0,C 180,E1 -7309.431,E2 -7309.431} C_VEL
LIN {X 0,Y 478.801,Z 987.903,A -85,B 0,C 180,E1 -7310.503,E2 -7310.503} C_VEL
LIN {X 0,Y 479.735,Z 976.103,A -85,B 0,C 180,E1 -7311.484,E2 -7311.484} C_VEL
LIN {X 0,Y 480.541,Z 964.068,A -85,B 0,C 180,E1 -7312.349,E2 -7312.349} C_VEL
LIN {X 0,Y 481.461,Z 951.186,A -85,B 0,C 180,E1 -7313.129,E2 -7313.129} C_VEL
LIN {X 0,Y 482.119,Z 939.191,A -85,B 0,C 180,E1 -7313.746,E2 -7313.746} C_VEL
LIN {X 0,Y 482.838,Z 926.505,A -85,B 0,C 180,E1 -7314.279,E2 -7314.279} C_VEL
LIN {X 0,Y 483.396,Z 912.834,A -85,B 0,C 180,E1 -7314.736,E2 -7314.736} C_VEL
LIN {X 0,Y 483.88,Z 900.169,A -85,B 0,C 180,E1 -7315.05,E2 -7315.05} C_VEL
LIN {X 0,Y 484.391,Z 874.876,A -85,B 0,C 180,E1 -7315.47,E2 -7315.47} C_VEL
LIN {X 0,Y 486.265,Z 721.475,A -85,B 0,C 180,E1 -7317.844,E2 -7317.844} C_VEL
LIN {X 0,Y 479.552,Z 693.959,A -85,B 0,C 180,E1 -7318.742,E2 -7318.742} C_VEL
LIN {X 0,Y 480.195,Z 681.949,A -85,B 0,C 180,E1 -7320.638,E2 -7320.638} C_VEL
LIN {X 0,Y 477.161,Z 669.02,A -85,B 0,C 180,E1 -7323.021,E2 -7323.021} C_VEL
LIN {X 0,Y 474.657,Z 659.264,A -85,B 0,C 180,E1 -7324.946,E2 -7324.946} C_VEL
LIN {X 0,Y 474.607,Z 659.172,A -85,B 0,C 180,E1 -7328.457,E2 -7328.457} C_VEL
LIN {X 0,Y 474.627,Z 659.167,A -85,B 0,C 180,E1 -7330.959,E2 -7330.959} C_VEL
LIN {X 0,Y 474.609,Z 659.164,A -85,B 0,C 180,E1 -7334.103,E2 -7334.103} C_VEL
LIN {X 0,Y 474.646,Z 659.173,A -85,B 0,C 180,E1 -7337.069,E2 -7337.069} C_VEL
LIN {X 0,Y 474.676,Z 659.167,A -85,B 0,C 180,E1 -7340.457,E2 -7340.457} C_VEL
LIN {X 0,Y 474.586,Z 659.166,A -85,B 0,C 180,E1 -7343.676,E2 -7343.676} C_VEL
LIN {X 0,Y 474.635,Z 659.172,A -85,B 0,C 180,E1 -7346.779,E2 -7346.779} C_VEL
LIN {X 0,Y 474.605,Z 659.162,A -85,B 0,C 180,E1 -7349.77,E2 -7349.77} C_VEL
LIN {X 0,Y 474.706,Z 659.151,A -85,B 0,C 180,E1 -7352.68,E2 -7352.68} C_VEL
LIN {X 0,Y 474.65,Z 659.169,A -85,B 0,C 180,E1 -7355.507,E2 -7355.507} C_VEL
LIN {X 0,Y 474.661,Z 659.169,A -85,B 0,C 180,E1 -7359.185,E2 -7359.185} C_VEL
LIN {X 0,Y 474.647,Z 659.164,A -85,B 0,C 180,E1 -7361.884,E2 -7361.884} C_VEL
LIN {X 0,Y 474.689,Z 659.169,A -85,B 0,C 180,E1 -7364.544,E2 -7364.544} C_VEL
LIN {X 0,Y 474.73,Z 659.154,A -85,B 0,C 180,E1 -7368.038,E2 -7368.038} C_VEL
LIN {X 0,Y 474.719,Z 659.152,A -85,B 0,C 180,E1 -7371.486,E2 -7371.486} C_VEL
LIN {X 0,Y 474.781,Z 659.151,A -85,B 0,C 180,E1 -7374.052,E2 -7374.052} C_VEL
LIN {X 0,Y 474.885,Z 659.136,A -85,B 0,C 180,E1 -7377.455,E2 -7377.455} C_VEL
LIN {X 0,Y 474.867,Z 659.143,A -85,B 0,C 180,E1 -7380.848,E2 -7380.848} C_VEL
LIN {X 0,Y 474.885,Z 659.129,A -85,B 0,C 180,E1 -7382.544,E2 -7382.544} C_VEL
LIN {X 0,Y 474.781,Z 659.153,A -85,B 0,C 180,E1 -7385.947,E2 -7385.947} C_VEL
LIN {X 0,Y 474.718,Z 659.156,A -85,B 0,C 180,E1 -7388.513,E2 -7388.513} C_VEL
LIN {X 0,Y 474.694,Z 659.16,A -85,B 0,C 180,E1 -7391.962,E2 -7391.962} C_VEL
LIN {X 0,Y 474.688,Z 659.165,A -85,B 0,C 180,E1 -7395.456,E2 -7395.456} C_VEL
LIN {X 0,Y 474.654,Z 659.167,A -85,B 0,C 180,E1 -7399.01,E2 -7399.01} C_VEL
LIN {X 0,Y 474.633,Z 659.171,A -85,B 0,C 180,E1 -7401.726,E2 -7401.726} C_VEL
LIN {X 0,Y 474.652,Z 659.175,A -85,B 0,C 180,E1 -7404.493,E2 -7404.493} C_VEL
LIN {X 0,Y 474.688,Z 659.149,A -85,B 0,C 180,E1 -7407.339,E2 -7407.339} C_VEL
LIN {X 0,Y 474.6,Z 659.171,A -85,B 0,C 180,E1 -7410.812,E2 -7410.812} C_VEL
LIN {X 0,Y 474.629,Z 659.17,A -85,B 0,C 180,E1 -7413.984,E2 -7413.984} C_VEL
LIN {X 0,Y 474.566,Z 659.163,A -85,B 0,C 180,E1 -7416.9,E2 -7416.9} C_VEL
LIN {X 0,Y 474.646,Z 659.171,A -85,B 0,C 180,E1 -7419.652,E2 -7419.652} C_VEL
LIN {X 0,Y 474.644,Z 659.177,A -85,B 0,C 180,E1 -7422.93,E2 -7422.93} C_VEL
LIN {X 0,Y 474.6,Z 659.177,A -85,B 0,C 180,E1 -7425.896,E2 -7425.896} C_VEL
LIN {X 0,Y 474.633,Z 659.176,A -85,B 0,C 180,E1 -7429.039,E2 -7429.039} C_VEL
LIN {X 0,Y 474.609,Z 659.18,A -85,B 0,C 180,E1 -7431.703,E2 -7431.703} C_VEL
LIN {X 0,Y 474.623,Z 659.174,A -85,B 0,C 180,E1 -7434.727,E2 -7434.727} C_VEL
LIN {X 0,Y 474.631,Z 659.179,A -85,B 0,C 180,E1 -7437.788,E2 -7437.788} C_VEL
LIN {X 0,Y 474.625,Z 659.174,A -85,B 0,C 180,E1 -7440.883,E2 -7440.883} C_VEL
LIN {X 0,Y 474.655,Z 659.175,A -85,B 0,C 180,E1 -7443.629,E2 -7443.629} C_VEL
LIN {X 0,Y 474.631,Z 659.175,A -85,B 0,C 180,E1 -7446.642,E2 -7446.642} C_VEL
LIN {X 0,Y 474.65,Z 659.176,A -85,B 0,C 180,E1 -7450.09,E2 -7450.09} C_VEL
LIN {X 0,Y 474.65,Z 659.173,A -85,B 0,C 180,E1 -7451.68,E2 -7451.68} C_VEL
LIN {X 0,Y 473.988,Z 659.259,A -85,B 0,C 180,E1 -7452.389,E2 -7452.389} C_VEL
LIN {X 0,Y 471.137,Z 659.615,A -85,B 0,C 180,E1 -7453.541,E2 -7453.541} C_VEL
LIN {X 0,Y 468.72,Z 659.914,A -85,B 0,C 180,E1 -7454.469,E2 -7454.469} C_VEL
LIN {X 0,Y 467.679,Z 660.041,A -85,B 0,C 180,E1 -7455.186,E2 -7455.186} C_VEL
LIN {X 0,Y 467.592,Z 660.051,A -85,B 0,C 180,E1 -7455.429,E2 -7455.429} C_VEL
LIN {X 0,Y 467.649,Z 660.046,A -85,B 0,C 180,E1 -7458.734,E2 -7458.734} C_VEL
LIN {X 0,Y 467.745,Z 660.035,A -85,B 0,C 180,E1 -7462.228,E2 -7462.228} C_VEL
LIN {X 0,Y 467.721,Z 660.039,A -85,B 0,C 180,E1 -7464.828,E2 -7464.828} C_VEL
LIN {X 0,Y 467.856,Z 660.02,A -85,B 0,C 180,E1 -7467.417,E2 -7467.417} C_VEL
LIN {X 0,Y 467.879,Z 660.016,A -85,B 0,C 180,E1 -7470,E2 -7470} C_VEL
LIN {X 0,Y 467.856,Z 660.02,A -85,B 0,C 180,E1 -7472.583,E2 -7472.583} C_VEL
LIN {X 0,Y 467.74,Z 660.033,A -85,B 0,C 180,E1 -7476.037,E2 -7476.037} C_VEL
LIN {X 0,Y 467.678,Z 660.041,A -85,B 0,C 180,E1 -7478.643,E2 -7478.643} C_VEL
LIN {X 0,Y 467.652,Z 660.044,A -85,B 0,C 180,E1 -7482.145,E2 -7482.145} C_VEL
LIN {X 0,Y 467.634,Z 660.049,A -85,B 0,C 180,E1 -7485.695,E2 -7485.695} C_VEL
LIN {X 0,Y 467.612,Z 660.049,A -85,B 0,C 180,E1 -7488.764,E2 -7488.764} C_VEL
LIN {X 0,Y 467.576,Z 660.054,A -85,B 0,C 180,E1 -7491.268,E2 -7491.268} C_VEL
LIN {X 0,Y 467.568,Z 660.058,A -85,B 0,C 180,E1 -7493.943,E2 -7493.943} C_VEL
LIN {X 0,Y 467.611,Z 660.049,A -85,B 0,C 180,E1 -7496.8,E2 -7496.8} C_VEL
LIN {X 0,Y 467.581,Z 660.055,A -85,B 0,C 180,E1 -7499.735,E2 -7499.735} C_VEL
LIN {X 0,Y 467.577,Z 660.055,A -85,B 0,C 180,E1 -7502.758,E2 -7502.758} C_VEL
LIN {X 0,Y 467.55,Z 660.056,A -85,B 0,C 180,E1 -7505.889,E2 -7505.889} C_VEL
LIN {X 0,Y 467.607,Z 660.049,A -85,B 0,C 180,E1 -7509.141,E2 -7509.141} C_VEL
LIN {X 0,Y 467.578,Z 660.056,A -85,B 0,C 180,E1 -7512.567,E2 -7512.567} C_VEL
LIN {X 0,Y 467.562,Z 660.058,A -85,B 0,C 180,E1 -7515.053,E2 -7515.053} C_VEL
LIN {X 0,Y 467.616,Z 660.049,A -85,B 0,C 180,E1 -7517.444,E2 -7517.444} C_VEL
LIN {X 0,Y 467.609,Z 660.053,A -85,B 0,C 180,E1 -7520.859,E2 -7520.859} C_VEL
LIN {X 0,Y 467.553,Z 660.032,A -85,B 0,C 180,E1 -7524.26,E2 -7524.26} C_VEL
LIN {X 0,Y 467.572,Z 660.059,A -85,B 0,C 180,E1 -7527.32,E2 -7527.32} C_VEL
LIN {X 0,Y 467.567,Z 660.029,A -85,B 0,C 180,E1 -7530.665,E2 -7530.665} C_VEL
LIN {X 0,Y 467.617,Z 660.033,A -85,B 0,C 180,E1 -7533.2,E2 -7533.2} C_VEL
LIN {X 0,Y 467.586,Z 660.047,A -85,B 0,C 180,E1 -7536.467,E2 -7536.467} C_VEL
LIN {X 0,Y 467.615,Z 660.052,A -85,B 0,C 180,E1 -7539.777,E2 -7539.777} C_VEL
LIN {X 0,Y 467.598,Z 660.043,A -85,B 0,C 180,E1 -7542.507,E2 -7542.507} C_VEL
LIN {X 0,Y 467.595,Z 660.047,A -85,B 0,C 180,E1 -7545.196,E2 -7545.196} C_VEL
LIN {X 0,Y 467.645,Z 660.034,A -85,B 0,C 180,E1 -7547.855,E2 -7547.855} C_VEL
LIN {X 0,Y 467.672,Z 660.032,A -85,B 0,C 180,E1 -7551.357,E2 -7551.357} C_VEL
LIN {X 0,Y 467.743,Z 660.028,A -85,B 0,C 180,E1 -7553.963,E2 -7553.963} C_VEL
LIN {X 0,Y 467.851,Z 660.005,A -85,B 0,C 180,E1 -7557.417,E2 -7557.417} C_VEL
LIN {X 0,Y 467.871,Z 660.014,A -85,B 0,C 180,E1 -7560,E2 -7560} C_VEL
LIN {X 0,Y 467.85,Z 660.012,A -85,B 0,C 180,E1 -7562.583,E2 -7562.583} C_VEL
LIN {X 0,Y 467.744,Z 660.028,A -85,B 0,C 180,E1 -7566.038,E2 -7566.038} C_VEL
LIN {X 0,Y 467.673,Z 660.03,A -85,B 0,C 180,E1 -7568.643,E2 -7568.643} C_VEL
LIN {X 0,Y 467.681,Z 660.031,A -85,B 0,C 180,E1 -7572.379,E2 -7572.379} C_VEL
LIN {X 0,Y 467.639,Z 660.042,A -85,B 0,C 180,E1 -7575.886,E2 -7575.886} C_VEL
LIN {X 0,Y 467.614,Z 660.047,A -85,B 0,C 180,E1 -7579.308,E2 -7579.308} C_VEL
LIN {X 0,Y 467.526,Z 660.05,A -85,B 0,C 180,E1 -7582.074,E2 -7582.074} C_VEL
LIN {X 0,Y 467.594,Z 660.049,A -85,B 0,C 180,E1 -7584.888,E2 -7584.888} C_VEL
LIN {X 0,Y 467.62,Z 660.022,A -85,B 0,C 180,E1 -7587.769,E2 -7587.769} C_VEL
LIN {X 0,Y 467.564,Z 660.046,A -85,B 0,C 180,E1 -7591.047,E2 -7591.047} C_VEL
LIN {X 0,Y 467.582,Z 660.043,A -85,B 0,C 180,E1 -7594.243,E2 -7594.243} C_VEL
LIN {X 0,Y 467.545,Z 660.05,A -85,B 0,C 180,E1 -7597.188,E2 -7597.188} C_VEL
LIN {X 0,Y 467.595,Z 660.041,A -85,B 0,C 180,E1 -7600.263,E2 -7600.263} C_VEL
LIN {X 0,Y 467.613,Z 660.046,A -85,B 0,C 180,E1 -7602.572,E2 -7602.572} C_VEL
LIN {X 0,Y 467.561,Z 660.044,A -85,B 0,C 180,E1 -7606.178,E2 -7606.178} C_VEL
LIN {X 0,Y 467.576,Z 660.046,A -85,B 0,C 180,E1 -7608.723,E2 -7608.723} C_VEL
LIN {X 0,Y 467.561,Z 660.035,A -85,B 0,C 180,E1 -7611.956,E2 -7611.956} C_VEL
LIN {X 0,Y 467.604,Z 660.134,A -85,B 0,C 180,E1 -7614.646,E2 -7614.646} C_VEL
LIN {X 0,Y 470.656,Z 671.863,A -85,B 0,C 180,E1 -7617.001,E2 -7617.001} C_VEL
LIN {X 0,Y 473.33,Z 683.308,A -85,B 0,C 180,E1 -7619.143,E2 -7619.143} C_VEL
LIN {X 0,Y 472.857,Z 693.589,A -85,B 0,C 180,E1 -7620.802,E2 -7620.802} C_VEL
LIN {X 0,Y 479.967,Z 722.908,A -85,B 0,C 180,E1 -7621.786,E2 -7621.786} C_VEL
LIN {X 0,Y 477.632,Z 896.014,A -85,B 0,C 180,E1 -7624.517,E2 -7624.517} C_VEL
LIN {X 0,Y 477.163,Z 907.732,A -85,B 0,C 180,E1 -7624.773,E2 -7624.773} C_VEL
LIN {X 0,Y 476.568,Z 921.073,A -85,B 0,C 180,E1 -7625.177,E2 -7625.177} C_VEL
LIN {X 0,Y 475.923,Z 934.198,A -85,B 0,C 180,E1 -7625.693,E2 -7625.693} C_VEL
LIN {X 0,Y 475.225,Z 945.589,A -85,B 0,C 180,E1 -7626.235,E2 -7626.235} C_VEL
LIN {X 0,Y 474.302,Z 959.337,A -85,B 0,C 180,E1 -7627.03,E2 -7627.03} C_VEL
LIN {X 0,Y 473.466,Z 970.137,A -85,B 0,C 180,E1 -7627.759,E2 -7627.759} C_VEL
LIN {X 0,Y 472.543,Z 982.581,A -85,B 0,C 180,E1 -7628.745,E2 -7628.745} C_VEL
LIN {X 0,Y 471.611,Z 993.802,A -85,B 0,C 180,E1 -7629.772,E2 -7629.772} C_VEL
LIN {X 0,Y 470.728,Z 1003.891,A -85,B 0,C 180,E1 -7630.825,E2 -7630.825} C_VEL
LIN {X 0,Y 469.946,Z 1013.166,A -85,B 0,C 180,E1 -7631.922,E2 -7631.922} C_VEL
LIN {X 0,Y 469.238,Z 1022.905,A -85,B 0,C 180,E1 -7633.243,E2 -7633.243} C_VEL
LIN {X 0,Y 468.608,Z 1031.432,A -85,B 0,C 180,E1 -7634.562,E2 -7634.562} C_VEL
LIN {X 0,Y 467.962,Z 1040.032,A -85,B 0,C 180,E1 -7636.097,E2 -7636.097} C_VEL
LIN {X 0,Y 467.594,Z 1046.464,A -85,B 0,C 180,E1 -7637.413,E2 -7637.413} C_VEL
LIN {X 0,Y 467.176,Z 1053.717,A -85,B 0,C 180,E1 -7639.162,E2 -7639.162} C_VEL
LIN {X 0,Y 466.932,Z 1058.361,A -85,B 0,C 180,E1 -7640.47,E2 -7640.47} C_VEL
LIN {X 0,Y 466.816,Z 1063.45,A -85,B 0,C 180,E1 -7642.213,E2 -7642.213} C_VEL
LIN {X 0,Y 466.708,Z 1067.437,A -85,B 0,C 180,E1 -7643.949,E2 -7643.949} C_VEL
LIN {X 0,Y 466.671,Z 1069.105,A -85,B 0,C 180,E1 -7644.816,E2 -7644.816} C_VEL
LIN {X 0,Y 466.639,Z 1071.562,A -85,B 0,C 180,E1 -7646.546,E2 -7646.546} C_VEL
LIN {X 0,Y 466.598,Z 1073.021,A -85,B 0,C 180,E1 -7648.274,E2 -7648.274} C_VEL
LIN {X 0,Y 466.594,Z 1073.505,A -85,B 0,C 180,E1 -7650,E2 -7650} C_VEL
LIN {X 0,Y 466.598,Z 1073.021,A -85,B 0,C 180,E1 -7651.726,E2 -7651.726} C_VEL
LIN {X 0,Y 466.639,Z 1071.562,A -85,B 0,C 180,E1 -7653.454,E2 -7653.454} C_VEL
LIN {X 0,Y 466.671,Z 1069.105,A -85,B 0,C 180,E1 -7655.184,E2 -7655.184} C_VEL
LIN {X 0,Y 466.787,Z 1065.621,A -85,B 0,C 180,E1 -7656.918,E2 -7656.918} C_VEL
LIN {X 0,Y 466.865,Z 1061.054,A -85,B 0,C 180,E1 -7658.658,E2 -7658.658} C_VEL
LIN {X 0,Y 467.1,Z 1055.337,A -85,B 0,C 180,E1 -7660.402,E2 -7660.402} C_VEL
LIN {X 0,Y 467.373,Z 1050.282,A -85,B 0,C 180,E1 -7661.712,E2 -7661.712} C_VEL
LIN {X 0,Y 467.743,Z 1043.364,A -85,B 0,C 180,E1 -7663.246,E2 -7663.246} C_VEL
LIN {X 0,Y 468.258,Z 1035.27,A -85,B 0,C 180,E1 -7664.782,E2 -7664.782} C_VEL
LIN {X 0,Y 468.862,Z 1027.755,A -85,B 0,C 180,E1 -7666.03,E2 -7666.03} C_VEL
LIN {X 0,Y 469.571,Z 1018.185,A -85,B 0,C 180,E1 -7667.417,E2 -7667.417} C_VEL
LIN {X 0,Y 470.26,Z 1009.613,A -85,B 0,C 180,E1 -7668.516,E2 -7668.516} C_VEL
LIN {X 0,Y 471.255,Z 997.791,A -85,B 0,C 180,E1 -7669.827,E2 -7669.827} C_VEL
LIN {X 0,Y 472.079,Z 987.695,A -85,B 0,C 180,E1 -7670.808,E2 -7670.808} C_VEL
LIN {X 0,Y 473.056,Z 975.895,A -85,B 0,C 180,E1 -7671.802,E2 -7671.802} C_VEL
LIN {X 0,Y 473.931,Z 963.861,A -85,B 0,C 180,E1 -7672.678,E2 -7672.678} C_VEL
LIN {X 0,Y 474.912,Z 950.94,A -85,B 0,C 180,E1 -7673.469,E2 -7673.469} C_VEL
LIN {X 0,Y 475.595,Z 938.984,A -85,B 0,C 180,E1 -7674.093,E2 -7674.093} C_VEL
LIN {X 0,Y 476.381,Z 925.552,A -85,B 0,C 180,E1 -7674.659,E2 -7674.659} C_VEL
LIN {X 0,Y 476.941,Z 912.628,A -85,B 0,C 180,E1 -7675.094,E2 -7675.094} C_VEL
LIN {X 0,Y 477.474,Z 898.878,A -85,B 0,C 180,E1 -7675.432,E2 -7675.432} C_VEL
LIN {X 0,Y 478.026,Z 870.89,A -85,B 0,C 180,E1 -7675.896,E2 -7675.896} C_VEL
LIN {X 0,Y 479.976,Z 722.76,A -85,B 0,C 180,E1 -7678.216,E2 -7678.216} C_VEL
LIN {X 0,Y 472.904,Z 693.735,A -85,B 0,C 180,E1 -7679.184,E2 -7679.184} C_VEL
LIN {X 0,Y 473.391,Z 685.032,A -85,B 0,C 180,E1 -7680.563,E2 -7680.563} C_VEL
LIN {X 0,Y 473.028,Z 681.944,A -85,B 0,C 180,E1 -7681.108,E2 -7681.108} C_VEL
LIN {X 0,Y 469.842,Z 668.734,A -85,B 0,C 180,E1 -7683.603,E2 -7683.603} C_VEL
LIN {X 0,Y 467.604,Z 660.137,A -85,B 0,C 180,E1 -7685.354,E2 -7685.354} C_VEL
LIN {X 0,Y 467.557,Z 660.052,A -85,B 0,C 180,E1 -7688.59,E2 -7688.59} C_VEL
LIN {X 0,Y 467.575,Z 660.047,A -85,B 0,C 180,E1 -7691.402,E2 -7691.402} C_VEL
LIN {X 0,Y 467.561,Z 660.044,A -85,B 0,C 180,E1 -7693.822,E2 -7693.822} C_VEL
LIN {X 0,Y 467.618,Z 660.045,A -85,B 0,C 180,E1 -7697.443,E2 -7697.443} C_VEL
LIN {X 0,Y 467.617,Z 660.046,A -85,B 0,C 180,E1 -7700.859,E2 -7700.859} C_VEL
LIN {X 0,Y 467.556,Z 660.038,A -85,B 0,C 180,E1 -7704.26,E2 -7704.26} C_VEL
LIN {X 0,Y 467.574,Z 660.052,A -85,B 0,C 180,E1 -7707.32,E2 -7707.32} C_VEL
LIN {X 0,Y 467.568,Z 660.022,A -85,B 0,C 180,E1 -7710.665,E2 -7710.665} C_VEL
LIN {X 0,Y 467.619,Z 660.037,A -85,B 0,C 180,E1 -7713.2,E2 -7713.2} C_VEL
LIN {X 0,Y 467.584,Z 660.049,A -85,B 0,C 180,E1 -7716.467,E2 -7716.467} C_VEL
LIN {X 0,Y 467.614,Z 660.046,A -85,B 0,C 180,E1 -7719.777,E2 -7719.777} C_VEL
LIN {X 0,Y 467.599,Z 660.044,A -85,B 0,C 180,E1 -7722.506,E2 -7722.506} C_VEL
LIN {X 0,Y 467.596,Z 660.048,A -85,B 0,C 180,E1 -7725.196,E2 -7725.196} C_VEL
LIN {X 0,Y 467.688,Z 660.031,A -85,B 0,C 180,E1 -7727.855,E2 -7727.855} C_VEL
LIN {X 0,Y 467.673,Z 660.031,A -85,B 0,C 180,E1 -7731.357,E2 -7731.357} C_VEL
LIN {X 0,Y 467.744,Z 660.028,A -85,B 0,C 180,E1 -7733.962,E2 -7733.962} C_VEL
LIN {X 0,Y 467.85,Z 660.012,A -85,B 0,C 180,E1 -7737.417,E2 -7737.417} C_VEL
LIN {X 0,Y 467.871,Z 660.014,A -85,B 0,C 180,E1 -7740,E2 -7740} C_VEL
LIN {X 0,Y 467.851,Z 660.005,A -85,B 0,C 180,E1 -7742.583,E2 -7742.583} C_VEL
LIN {X 0,Y 467.743,Z 660.029,A -85,B 0,C 180,E1 -7746.037,E2 -7746.037} C_VEL
LIN {X 0,Y 467.672,Z 660.034,A -85,B 0,C 180,E1 -7748.643,E2 -7748.643} C_VEL
LIN {X 0,Y 467.645,Z 660.035,A -85,B 0,C 180,E1 -7752.145,E2 -7752.145} C_VEL
LIN {X 0,Y 467.628,Z 660.048,A -85,B 0,C 180,E1 -7755.695,E2 -7755.695} C_VEL
LIN {X 0,Y 467.606,Z 660.046,A -85,B 0,C 180,E1 -7758.765,E2 -7758.765} C_VEL
LIN {X 0,Y 467.604,Z 660.044,A -85,B 0,C 180,E1 -7761.279,E2 -7761.279} C_VEL
LIN {X 0,Y 467.567,Z 660.052,A -85,B 0,C 180,E1 -7763.943,E2 -7763.943} C_VEL
LIN {X 0,Y 467.617,Z 660.033,A -85,B 0,C 180,E1 -7766.8,E2 -7766.8} C_VEL
LIN {X 0,Y 467.576,Z 660.031,A -85,B 0,C 180,E1 -7769.736,E2 -7769.736} C_VEL
LIN {X 0,Y 467.574,Z 660.057,A -85,B 0,C 180,E1 -7772.759,E2 -7772.759} C_VEL
LIN {X 0,Y 467.547,Z 660.032,A -85,B 0,C 180,E1 -7775.89,E2 -7775.89} C_VEL
LIN {X 0,Y 467.609,Z 660.053,A -85,B 0,C 180,E1 -7779.141,E2 -7779.141} C_VEL
LIN {X 0,Y 467.61,Z 660.05,A -85,B 0,C 180,E1 -7782.572,E2 -7782.572} C_VEL
LIN {X 0,Y 467.562,Z 660.06,A -85,B 0,C 180,E1 -7785.054,E2 -7785.054} C_VEL
LIN {X 0,Y 467.58,Z 660.056,A -85,B 0,C 180,E1 -7787.44,E2 -7787.44} C_VEL
LIN {X 0,Y 467.607,Z 660.049,A -85,B 0,C 180,E1 -7790.859,E2 -7790.859} C_VEL
LIN {X 0,Y 467.556,Z 660.055,A -85,B 0,C 180,E1 -7794.261,E2 -7794.261} C_VEL
LIN {X 0,Y 467.576,Z 660.055,A -85,B 0,C 180,E1 -7797.321,E2 -7797.321} C_VEL
LIN {X 0,Y 467.571,Z 660.053,A -85,B 0,C 180,E1 -7800.666,E2 -7800.666} C_VEL
LIN {X 0,Y 467.61,Z 660.049,A -85,B 0,C 180,E1 -7803.2,E2 -7803.2} C_VEL
LIN {X 0,Y 467.588,Z 660.053,A -85,B 0,C 180,E1 -7806.468,E2 -7806.468} C_VEL
LIN {X 0,Y 467.618,Z 660.049,A -85,B 0,C 180,E1 -7809.778,E2 -7809.778} C_VEL
LIN {X 0,Y 467.604,Z 660.054,A -85,B 0,C 180,E1 -7812.507,E2 -7812.507} C_VEL
LIN {X 0,Y 467.592,Z 660.051,A -85,B 0,C 180,E1 -7815.429,E2 -7815.429} C_VEL
LIN {X 0,Y 466.922,Z 660.138,A -85,B 0,C 180,E1 -7816.148,E2 -7816.148} C_VEL
LIN {X 0,Y 464.079,Z 660.488,A -85,B 0,C 180,E1 -7817.317,E2 -7817.317} C_VEL
LIN {X 0,Y 461.68,Z 660.792,A -85,B 0,C 180,E1 -7818.259,E2 -7818.259} C_VEL
LIN {X 0,Y 460.654,Z 660.918,A -85,B 0,C 180,E1 -7818.986,E2 -7818.986} C_VEL
LIN {X 0,Y 460.573,Z 660.925,A -85,B 0,C 180,E1 -7819.233,E2 -7819.233} C_VEL
LIN {X 0,Y 460.716,Z 660.91,A -85,B 0,C 180,E1 -7822.538,E2 -7822.538} C_VEL
LIN {X 0,Y 460.694,Z 660.915,A -85,B 0,C 180,E1 -7824.748,E2 -7824.748} C_VEL
LIN {X 0,Y 460.821,Z 660.896,A -85,B 0,C 180,E1 -7827.378,E2 -7827.378} C_VEL
LIN {X 0,Y 460.85,Z 660.892,A -85,B 0,C 180,E1 -7830,E2 -7830} C_VEL
LIN {X 0,Y 460.821,Z 660.897,A -85,B 0,C 180,E1 -7832.622,E2 -7832.622} C_VEL
LIN {X 0,Y 460.706,Z 660.909,A -85,B 0,C 180,E1 -7836.13,E2 -7836.13} C_VEL
LIN {X 0,Y 460.625,Z 660.92,A -85,B 0,C 180,E1 -7838.776,E2 -7838.776} C_VEL
LIN {X 0,Y 460.609,Z 660.92,A -85,B 0,C 180,E1 -7842.445,E2 -7842.445} C_VEL
LIN {X 0,Y 460.595,Z 660.925,A -85,B 0,C 180,E1 -7845.997,E2 -7845.997} C_VEL
LIN {X 0,Y 460.566,Z 660.927,A -85,B 0,C 180,E1 -7848.901,E2 -7848.901} C_VEL
LIN {X 0,Y 460.511,Z 660.936,A -85,B 0,C 180,E1 -7851.485,E2 -7851.485} C_VEL
LIN {X 0,Y 460.537,Z 660.932,A -85,B 0,C 180,E1 -7854.332,E2 -7854.332} C_VEL
LIN {X 0,Y 460.574,Z 660.925,A -85,B 0,C 180,E1 -7857.243,E2 -7857.243} C_VEL
LIN {X 0,Y 460.521,Z 660.935,A -85,B 0,C 180,E1 -7860.238,E2 -7860.238} C_VEL
LIN {X 0,Y 460.523,Z 660.931,A -85,B 0,C 180,E1 -7863.324,E2 -7863.324} C_VEL
LIN {X 0,Y 460.472,Z 660.942,A -85,B 0,C 180,E1 -7866.529,E2 -7866.529} C_VEL
LIN {X 0,Y 460.567,Z 660.925,A -85,B 0,C 180,E1 -7869.857,E2 -7869.857} C_VEL
LIN {X 0,Y 460.505,Z 660.938,A -85,B 0,C 180,E1 -7872.9,E2 -7872.9} C_VEL
LIN {X 0,Y 460.515,Z 660.931,A -85,B 0,C 180,E1 -7875.828,E2 -7875.828} C_VEL
LIN {X 0,Y 460.535,Z 660.935,A -85,B 0,C 180,E1 -7878.99,E2 -7878.99} C_VEL
LIN {X 0,Y 460.538,Z 660.928,A -85,B 0,C 180,E1 -7881.269,E2 -7881.269} C_VEL
LIN {X 0,Y 460.504,Z 660.91,A -85,B 0,C 180,E1 -7884.554,E2 -7884.554} C_VEL
LIN {X 0,Y 460.522,Z 660.932,A -85,B 0,C 180,E1 -7887.715,E2 -7887.715} C_VEL
LIN {X 0,Y 460.536,Z 660.902,A -85,B 0,C 180,E1 -7890.769,E2 -7890.769} C_VEL
LIN {X 0,Y 460.558,Z 660.921,A -85,B 0,C 180,E1 -7893.735,E2 -7893.735} C_VEL
LIN {X 0,Y 460.541,Z 660.924,A -85,B 0,C 180,E1 -7896.624,E2 -7896.624} C_VEL
LIN {X 0,Y 460.562,Z 660.925,A -85,B 0,C 180,E1 -7899.454,E2 -7899.454} C_VEL
LIN {X 0,Y 460.548,Z 660.921,A -85,B 0,C 180,E1 -7902.23,E2 -7902.23} C_VEL
LIN {X 0,Y 460.554,Z 660.924,A -85,B 0,C 180,E1 -7904.965,E2 -7904.965} C_VEL
LIN {X 0,Y 460.602,Z 660.921,A -85,B 0,C 180,E1 -7908.559,E2 -7908.559} C_VEL
LIN {X 0,Y 460.684,Z 660.904,A -85,B 0,C 180,E1 -7912.109,E2 -7912.109} C_VEL
LIN {X 0,Y 460.696,Z 660.91,A -85,B 0,C 180,E1 -7914.749,E2 -7914.749} C_VEL
LIN {X 0,Y 460.816,Z 660.881,A -85,B 0,C 180,E1 -7917.378,E2 -7917.378} C_VEL
LIN {X 0,Y 460.842,Z 660.89,A -85,B 0,C 180,E1 -7920,E2 -7920} C_VEL
LIN {X 0,Y 460.816,Z 660.888,A -85,B 0,C 180,E1 -7922.623,E2 -7922.623} C_VEL
LIN {X 0,Y 460.708,Z 660.905,A -85,B 0,C 180,E1 -7926.13,E2 -7926.13} C_VEL
LIN {X 0,Y 460.62,Z 660.909,A -85,B 0,C 180,E1 -7928.776,E2 -7928.776} C_VEL
LIN {X 0,Y 460.624,Z 660.911,A -85,B 0,C 180,E1 -7932.457,E2 -7932.457} C_VEL
LIN {X 0,Y 460.59,Z 660.919,A -85,B 0,C 180,E1 -7935.998,E2 -7935.998} C_VEL
LIN {X 0,Y 460.561,Z 660.92,A -85,B 0,C 180,E1 -7938.902,E2 -7938.902} C_VEL
LIN {X 0,Y 460.506,Z 660.931,A -85,B 0,C 180,E1 -7941.486,E2 -7941.486} C_VEL
LIN {X 0,Y 460.534,Z 660.929,A -85,B 0,C 180,E1 -7944.333,E2 -7944.333} C_VEL
LIN {X 0,Y 460.575,Z 660.909,A -85,B 0,C 180,E1 -7947.244,E2 -7947.244} C_VEL
LIN {X 0,Y 460.519,Z 660.914,A -85,B 0,C 180,E1 -7950.239,E2 -7950.239} C_VEL
LIN {X 0,Y 460.522,Z 660.931,A -85,B 0,C 180,E1 -7953.325,E2 -7953.325} C_VEL
LIN {X 0,Y 460.472,Z 660.924,A -85,B 0,C 180,E1 -7956.53,E2 -7956.53} C_VEL
LIN {X 0,Y 460.578,Z 660.922,A -85,B 0,C 180,E1 -7959.858,E2 -7959.858} C_VEL
LIN {X 0,Y 460.537,Z 660.931,A -85,B 0,C 180,E1 -7962.905,E2 -7962.905} C_VEL
LIN {X 0,Y 460.513,Z 660.919,A -85,B 0,C 180,E1 -7965.83,E2 -7965.83} C_VEL
LIN {X 0,Y 460.528,Z 660.922,A -85,B 0,C 180,E1 -7968.99,E2 -7968.99} C_VEL
LIN {X 0,Y 460.521,Z 660.929,A -85,B 0,C 180,E1 -7971.268,E2 -7971.268} C_VEL
LIN {X 0,Y 460.543,Z 661.055,A -85,B 0,C 180,E1 -7974.24,E2 -7974.24} C_VEL
LIN {X 0,Y 463.716,Z 673.221,A -85,B 0,C 180,E1 -7976.73,E2 -7976.73} C_VEL
LIN {X 0,Y 466.472,Z 684.781,A -85,B 0,C 180,E1 -7978.936,E2 -7978.936} C_VEL
LIN {X 0,Y 466.306,Z 690.643,A -85,B 0,C 180,E1 -7979.926,E2 -7979.926} C_VEL
LIN {X 0,Y 466.182,Z 693.434,A -85,B 0,C 180,E1 -7980.35,E2 -7980.35} C_VEL
LIN {X 0,Y 473.567,Z 723.564,A -85,B 0,C 180,E1 -7981.384,E2 -7981.384} C_VEL
LIN {X 0,Y 473.45,Z 743.306,A -85,B 0,C 180,E1 -7981.709,E2 -7981.709} C_VEL
LIN {X 0,Y 471.204,Z 896.156,A -85,B 0,C 180,E1 -7984.152,E2 -7984.152} C_VEL
LIN {X 0,Y 470.706,Z 908.506,A -85,B 0,C 180,E1 -7984.432,E2 -7984.432} C_VEL
LIN {X 0,Y 470.07,Z 921.613,A -85,B 0,C 180,E1 -7984.839,E2 -7984.839} C_VEL
LIN {X 0,Y 469.439,Z 933.992,A -85,B 0,C 180,E1 -7985.335,E2 -7985.335} C_VEL
LIN {X 0,Y 468.686,Z 945.382,A -85,B 0,C 180,E1 -7985.883,E2 -7985.883} C_VEL
LIN {X 0,Y 467.819,Z 957.887,A -85,B 0,C 180,E1 -7986.606,E2 -7986.606} C_VEL
LIN {X 0,Y 466.851,Z 969.93,A -85,B 0,C 180,E1 -7987.427,E2 -7987.427} C_VEL
LIN {X 0,Y 465.854,Z 982.374,A -85,B 0,C 180,E1 -7988.425,E2 -7988.425} C_VEL
LIN {X 0,Y 464.91,Z 993.18,A -85,B 0,C 180,E1 -7989.423,E2 -7989.423} C_VEL
LIN {X 0,Y 463.882,Z 1003.682,A -85,B 0,C 180,E1 -7990.531,E2 -7990.531} C_VEL
LIN {X 0,Y 463.117,Z 1012.958,A -85,B 0,C 180,E1 -7991.646,E2 -7991.646} C_VEL
LIN {X 0,Y 462.335,Z 1022.696,A -85,B 0,C 180,E1 -7992.986,E2 -7992.986} C_VEL
LIN {X 0,Y 461.642,Z 1031.223,A -85,B 0,C 180,E1 -7994.323,E2 -7994.323} C_VEL
LIN {X 0,Y 460.965,Z 1039.823,A -85,B 0,C 180,E1 -7995.881,E2 -7995.881} C_VEL
LIN {X 0,Y 460.545,Z 1046.255,A -85,B 0,C 180,E1 -7997.217,E2 -7997.217} C_VEL
LIN {X 0,Y 460.133,Z 1053.509,A -85,B 0,C 180,E1 -7998.994,E2 -7998.994} C_VEL
LIN {X 0,Y 459.859,Z 1058.153,A -85,B 0,C 180,E1 -8000.322,E2 -8000.322} C_VEL
LIN {X 0,Y 459.728,Z 1063.243,A -85,B 0,C 180,E1 -8002.092,E2 -8002.092} C_VEL
LIN {X 0,Y 459.636,Z 1067.231,A -85,B 0,C 180,E1 -8003.856,E2 -8003.856} C_VEL
LIN {X 0,Y 459.523,Z 1070.174,A -85,B 0,C 180,E1 -8005.614,E2 -8005.614} C_VEL
LIN {X 0,Y 459.535,Z 1071.356,A -85,B 0,C 180,E1 -8006.493,E2 -8006.493} C_VEL
LIN {X 0,Y 459.511,Z 1072.816,A -85,B 0,C 180,E1 -8008.247,E2 -8008.247} C_VEL
LIN {X 0,Y 459.526,Z 1073.301,A -85,B 0,C 180,E1 -8010,E2 -8010} C_VEL
LIN {X 0,Y 459.511,Z 1072.816,A -85,B 0,C 180,E1 -8011.753,E2 -8011.753} C_VEL
LIN {X 0,Y 459.535,Z 1071.356,A -85,B 0,C 180,E1 -8013.507,E2 -8013.507} C_VEL
LIN {X 0,Y 459.583,Z 1068.899,A -85,B 0,C 180,E1 -8015.264,E2 -8015.264} C_VEL
LIN {X 0,Y 459.709,Z 1065.415,A -85,B 0,C 180,E1 -8017.025,E2 -8017.025} C_VEL
LIN {X 0,Y 459.802,Z 1060.847,A -85,B 0,C 180,E1 -8018.792,E2 -8018.792} C_VEL
LIN {X 0,Y 460.034,Z 1055.129,A -85,B 0,C 180,E1 -8020.563,E2 -8020.563} C_VEL
LIN {X 0,Y 460.348,Z 1050.075,A -85,B 0,C 180,E1 -8021.894,E2 -8021.894} C_VEL
LIN {X 0,Y 460.783,Z 1042.044,A -85,B 0,C 180,E1 -8023.674,E2 -8023.674} C_VEL
LIN {X 0,Y 461.303,Z 1035.062,A -85,B 0,C 180,E1 -8025.01,E2 -8025.01} C_VEL
LIN {X 0,Y 461.947,Z 1026.45,A -85,B 0,C 180,E1 -8026.446,E2 -8026.446} C_VEL
LIN {X 0,Y 462.678,Z 1017.976,A -85,B 0,C 180,E1 -8027.685,E2 -8027.685} C_VEL
LIN {X 0,Y 463.431,Z 1009.405,A -85,B 0,C 180,E1 -8028.799,E2 -8028.799} C_VEL
LIN {X 0,Y 464.522,Z 997.309,A -85,B 0,C 180,E1 -8030.156,E2 -8030.156} C_VEL
LIN {X 0,Y 465.48,Z 986.115,A -85,B 0,C 180,E1 -8031.245,E2 -8031.245} C_VEL
LIN {X 0,Y 466.391,Z 975.687,A -85,B 0,C 180,E1 -8032.13,E2 -8032.13} C_VEL
LIN {X 0,Y 467.332,Z 963.654,A -85,B 0,C 180,E1 -8033.016,E2 -8033.016} C_VEL
LIN {X 0,Y 468.324,Z 951.17,A -85,B 0,C 180,E1 -8033.794,E2 -8033.794} C_VEL
LIN {X 0,Y 469.101,Z 938.778,A -85,B 0,C 180,E1 -8034.448,E2 -8034.448} C_VEL
LIN {X 0,Y 469.935,Z 925.347,A -85,B 0,C 180,E1 -8035.02,E2 -8035.02} C_VEL
LIN {X 0,Y 470.511,Z 912.423,A -85,B 0,C 180,E1 -8035.461,E2 -8035.461} C_VEL
LIN {X 0,Y 471.053,Z 898.949,A -85,B 0,C 180,E1 -8035.798,E2 -8035.798} C_VEL
LIN {X 0,Y 471.576,Z 875.352,A -85,B 0,C 180,E1 -8036.199,E2 -8036.199} C_VEL
LIN {X 0,Y 473.709,Z 724.013,A -85,B 0,C 180,E1 -8038.599,E2 -8038.599} C_VEL
LIN {X 0,Y 466.253,Z 693.608,A -85,B 0,C 180,E1 -8039.634,E2 -8039.634} C_VEL
LIN {X 0,Y 466.485,Z 689.183,A -85,B 0,C 180,E1 -8040.311,E2 -8040.311} C_VEL
LIN {X 0,Y 466.471,Z 684.781,A -85,B 0,C 180,E1 -8041.064,E2 -8041.064} C_VEL
LIN {X 0,Y 463.119,Z 670.819,A -85,B 0,C 180,E1 -8043.74,E2 -8043.74} C_VEL
LIN {X 0,Y 460.543,Z 661.051,A -85,B 0,C 180,E1 -8045.76,E2 -8045.76} C_VEL
LIN {X 0,Y 460.54,Z 660.928,A -85,B 0,C 180,E1 -8048.897,E2 -8048.897} C_VEL
LIN {X 0,Y 460.518,Z 660.933,A -85,B 0,C 180,E1 -8052.181,E2 -8052.181} C_VEL
LIN {X 0,Y 460.516,Z 660.924,A -85,B 0,C 180,E1 -8055.411,E2 -8055.411} C_VEL
LIN {X 0,Y 460.54,Z 660.914,A -85,B 0,C 180,E1 -8058.395,E2 -8058.395} C_VEL
LIN {X 0,Y 460.542,Z 660.929,A -85,B 0,C 180,E1 -8061.269,E2 -8061.269} C_VEL
LIN {X 0,Y 460.506,Z 660.916,A -85,B 0,C 180,E1 -8064.554,E2 -8064.554} C_VEL
LIN {X 0,Y 460.525,Z 660.933,A -85,B 0,C 180,E1 -8067.715,E2 -8067.715} C_VEL
LIN {X 0,Y 460.538,Z 660.895,A -85,B 0,C 180,E1 -8070.769,E2 -8070.769} C_VEL
LIN {X 0,Y 460.559,Z 660.918,A -85,B 0,C 180,E1 -8073.734,E2 -8073.734} C_VEL
LIN {X 0,Y 460.537,Z 660.924,A -85,B 0,C 180,E1 -8076.623,E2 -8076.623} C_VEL
LIN {X 0,Y 460.542,Z 660.927,A -85,B 0,C 180,E1 -8079.452,E2 -8079.452} C_VEL
LIN {X 0,Y 460.549,Z 660.921,A -85,B 0,C 180,E1 -8082.23,E2 -8082.23} C_VEL
LIN {X 0,Y 460.555,Z 660.928,A -85,B 0,C 180,E1 -8084.964,E2 -8084.964} C_VEL
LIN {X 0,Y 460.647,Z 660.908,A -85,B 0,C 180,E1 -8087.667,E2 -8087.667} C_VEL
LIN {X 0,Y 460.62,Z 660.91,A -85,B 0,C 180,E1 -8091.224,E2 -8091.224} C_VEL
LIN {X 0,Y 460.708,Z 660.904,A -85,B 0,C 180,E1 -8093.87,E2 -8093.87} C_VEL
LIN {X 0,Y 460.816,Z 660.887,A -85,B 0,C 180,E1 -8097.377,E2 -8097.377} C_VEL
LIN {X 0,Y 460.842,Z 660.889,A -85,B 0,C 180,E1 -8100,E2 -8100} C_VEL
LIN {X 0,Y 460.816,Z 660.881,A -85,B 0,C 180,E1 -8102.622,E2 -8102.622} C_VEL
LIN {X 0,Y 460.707,Z 660.904,A -85,B 0,C 180,E1 -8106.13,E2 -8106.13} C_VEL
LIN {X 0,Y 460.619,Z 660.912,A -85,B 0,C 180,E1 -8108.776,E2 -8108.776} C_VEL
LIN {X 0,Y 460.602,Z 660.909,A -85,B 0,C 180,E1 -8112.445,E2 -8112.445} C_VEL
LIN {X 0,Y 460.589,Z 660.924,A -85,B 0,C 180,E1 -8115.998,E2 -8115.998} C_VEL
LIN {X 0,Y 460.56,Z 660.923,A -85,B 0,C 180,E1 -8118.902,E2 -8118.902} C_VEL
LIN {X 0,Y 460.554,Z 660.923,A -85,B 0,C 180,E1 -8121.483,E2 -8121.483} C_VEL
LIN {X 0,Y 460.535,Z 660.934,A -85,B 0,C 180,E1 -8124.332,E2 -8124.332} C_VEL
LIN {X 0,Y 460.573,Z 660.906,A -85,B 0,C 180,E1 -8127.243,E2 -8127.243} C_VEL
LIN {X 0,Y 460.516,Z 660.913,A -85,B 0,C 180,E1 -8130.239,E2 -8130.239} C_VEL
LIN {X 0,Y 460.519,Z 660.929,A -85,B 0,C 180,E1 -8133.325,E2 -8133.325} C_VEL
LIN {X 0,Y 460.469,Z 660.913,A -85,B 0,C 180,E1 -8136.529,E2 -8136.529} C_VEL
LIN {X 0,Y 460.569,Z 660.924,A -85,B 0,C 180,E1 -8139.858,E2 -8139.858} C_VEL
LIN {X 0,Y 460.534,Z 660.934,A -85,B 0,C 180,E1 -8142.905,E2 -8142.905} C_VEL
LIN {X 0,Y 460.503,Z 660.934,A -85,B 0,C 180,E1 -8145.831,E2 -8145.831} C_VEL
LIN {X 0,Y 460.531,Z 660.932,A -85,B 0,C 180,E1 -8148.99,E2 -8148.99} C_VEL
LIN {X 0,Y 460.536,Z 660.934,A -85,B 0,C 180,E1 -8151.269,E2 -8151.269} C_VEL
LIN {X 0,Y 460.507,Z 660.932,A -85,B 0,C 180,E1 -8154.555,E2 -8154.555} C_VEL
LIN {X 0,Y 460.526,Z 660.936,A -85,B 0,C 180,E1 -8157.716,E2 -8157.716} C_VEL
LIN {X 0,Y 460.54,Z 660.929,A -85,B 0,C 180,E1 -8160.77,E2 -8160.77} C_VEL
LIN {X 0,Y 460.557,Z 660.931,A -85,B 0,C 180,E1 -8163.735,E2 -8163.735} C_VEL
LIN {X 0,Y 460.541,Z 660.93,A -85,B 0,C 180,E1 -8166.624,E2 -8166.624} C_VEL
LIN {X 0,Y 460.546,Z 660.929,A -85,B 0,C 180,E1 -8169.453,E2 -8169.453} C_VEL
LIN {X 0,Y 460.554,Z 660.93,A -85,B 0,C 180,E1 -8172.23,E2 -8172.23} C_VEL
LIN {X 0,Y 460.561,Z 660.93,A -85,B 0,C 180,E1 -8174.965,E2 -8174.965} C_VEL
LIN {X 0,Y 460.607,Z 660.924,A -85,B 0,C 180,E1 -8178.559,E2 -8178.559} C_VEL
LIN {X 0,Y 460.573,Z 660.925,A -85,B 0,C 180,E1 -8179.233,E2 -8179.233} C_VEL
LIN {X 0,Y 459.918,Z 661.009,A -85,B 0,C 180,E1 -8179.963,E2 -8179.963} C_VEL
LIN {X 0,Y 457.101,Z 661.363,A -85,B 0,C 180,E1 -8181.15,E2 -8181.15} C_VEL
LIN {X 0,Y 454.722,Z 661.659,A -85,B 0,C 180,E1 -8182.107,E2 -8182.107} C_VEL
LIN {X 0,Y 453.71,Z 661.783,A -85,B 0,C 180,E1 -8182.846,E2 -8182.846} C_VEL
LIN {X 0,Y 453.633,Z 661.791,A -85,B 0,C 180,E1 -8183.096,E2 -8183.096} C_VEL
LIN {X 0,Y 453.667,Z 661.79,A -85,B 0,C 180,E1 -8184.667,E2 -8184.667} C_VEL
LIN {X 0,Y 453.762,Z 661.776,A -85,B 0,C 180,E1 -8187.337,E2 -8187.337} C_VEL
LIN {X 0,Y 453.82,Z 661.768,A -85,B 0,C 180,E1 -8190,E2 -8190} C_VEL
LIN {X 0,Y 453.762,Z 661.777,A -85,B 0,C 180,E1 -8192.663,E2 -8192.663} C_VEL
LIN {X 0,Y 453.674,Z 661.785,A -85,B 0,C 180,E1 -8196.225,E2 -8196.225} C_VEL
LIN {X 0,Y 453.588,Z 661.797,A -85,B 0,C 180,E1 -8198.913,E2 -8198.913} C_VEL
LIN {X 0,Y 453.559,Z 661.799,A -85,B 0,C 180,E1 -8202.529,E2 -8202.529} C_VEL
LIN {X 0,Y 453.54,Z 661.802,A -85,B 0,C 180,E1 -8206.196,E2 -8206.196} C_VEL
LIN {X 0,Y 453.515,Z 661.806,A -85,B 0,C 180,E1 -8209.04,E2 -8209.04} C_VEL
LIN {X 0,Y 453.472,Z 661.813,A -85,B 0,C 180,E1 -8211.836,E2 -8211.836} C_VEL
LIN {X 0,Y 453.509,Z 661.806,A -85,B 0,C 180,E1 -8214.734,E2 -8214.734} C_VEL
LIN {X 0,Y 453.533,Z 661.806,A -85,B 0,C 180,E1 -8217.961,E2 -8217.961} C_VEL
LIN {X 0,Y 453.477,Z 661.811,A -85,B 0,C 180,E1 -8220.759,E2 -8220.759} C_VEL
LIN {X 0,Y 453.471,Z 661.813,A -85,B 0,C 180,E1 -8223.912,E2 -8223.912} C_VEL
LIN {X 0,Y 453.464,Z 661.811,A -85,B 0,C 180,E1 -8227.187,E2 -8227.187} C_VEL
LIN {X 0,Y 453.523,Z 661.802,A -85,B 0,C 180,E1 -8229.445,E2 -8229.445} C_VEL
LIN {X 0,Y 453.455,Z 661.816,A -85,B 0,C 180,E1 -8232.994,E2 -8232.994} C_VEL
LIN {X 0,Y 453.468,Z 661.809,A -85,B 0,C 180,E1 -8235.78,E2 -8235.78} C_VEL
LIN {X 0,Y 453.488,Z 661.807,A -85,B 0,C 180,E1 -8238.211,E2 -8238.211} C_VEL
LIN {X 0,Y 453.523,Z 661.807,A -85,B 0,C 180,E1 -8240.787,E2 -8240.787} C_VEL
LIN {X 0,Y 453.447,Z 661.785,A -85,B 0,C 180,E1 -8243.917,E2 -8243.917} C_VEL
LIN {X 0,Y 453.473,Z 661.812,A -85,B 0,C 180,E1 -8247.151,E2 -8247.151} C_VEL
LIN {X 0,Y 453.504,Z 661.782,A -85,B 0,C 180,E1 -8250.271,E2 -8250.271} C_VEL
LIN {X 0,Y 453.503,Z 661.791,A -85,B 0,C 180,E1 -8253.294,E2 -8253.294} C_VEL
LIN {X 0,Y 453.497,Z 661.803,A -85,B 0,C 180,E1 -8256.239,E2 -8256.239} C_VEL
LIN {X 0,Y 453.507,Z 661.801,A -85,B 0,C 180,E1 -8259.119,E2 -8259.119} C_VEL
LIN {X 0,Y 453.5,Z 661.799,A -85,B 0,C 180,E1 -8261.944,E2 -8261.944} C_VEL
LIN {X 0,Y 453.528,Z 661.8,A -85,B 0,C 180,E1 -8264.726,E2 -8264.726} C_VEL
LIN {X 0,Y 453.551,Z 661.797,A -85,B 0,C 180,E1 -8268.379,E2 -8268.379} C_VEL
LIN {X 0,Y 453.641,Z 661.781,A -85,B 0,C 180,E1 -8271.985,E2 -8271.985} C_VEL
LIN {X 0,Y 453.669,Z 661.787,A -85,B 0,C 180,E1 -8274.667,E2 -8274.667} C_VEL
LIN {X 0,Y 453.756,Z 661.761,A -85,B 0,C 180,E1 -8277.337,E2 -8277.337} C_VEL
LIN {X 0,Y 453.813,Z 661.766,A -85,B 0,C 180,E1 -8280,E2 -8280} C_VEL
LIN {X 0,Y 453.756,Z 661.767,A -85,B 0,C 180,E1 -8282.663,E2 -8282.663} C_VEL
LIN {X 0,Y 453.674,Z 661.782,A -85,B 0,C 180,E1 -8286.226,E2 -8286.226} C_VEL
LIN {X 0,Y 453.584,Z 661.788,A -85,B 0,C 180,E1 -8288.914,E2 -8288.914} C_VEL
LIN {X 0,Y 453.592,Z 661.787,A -85,B 0,C 180,E1 -8292.551,E2 -8292.551} C_VEL
LIN {X 0,Y 453.535,Z 661.797,A -85,B 0,C 180,E1 -8296.196,E2 -8296.196} C_VEL
LIN {X 0,Y 453.51,Z 661.8,A -85,B 0,C 180,E1 -8299.041,E2 -8299.041} C_VEL
LIN {X 0,Y 453.467,Z 661.803,A -85,B 0,C 180,E1 -8301.837,E2 -8301.837} C_VEL
LIN {X 0,Y 453.505,Z 661.804,A -85,B 0,C 180,E1 -8304.735,E2 -8304.735} C_VEL
LIN {X 0,Y 453.53,Z 661.771,A -85,B 0,C 180,E1 -8307.962,E2 -8307.962} C_VEL
LIN {X 0,Y 453.475,Z 661.8,A -85,B 0,C 180,E1 -8310.76,E2 -8310.76} C_VEL
LIN {X 0,Y 453.47,Z 661.805,A -85,B 0,C 180,E1 -8313.913,E2 -8313.913} C_VEL
LIN {X 0,Y 453.465,Z 661.803,A -85,B 0,C 180,E1 -8317.188,E2 -8317.188} C_VEL
LIN {X 0,Y 453.53,Z 661.801,A -85,B 0,C 180,E1 -8319.446,E2 -8319.446} C_VEL
LIN {X 0,Y 453.486,Z 661.809,A -85,B 0,C 180,E1 -8322.992,E2 -8322.992} C_VEL
LIN {X 0,Y 453.467,Z 661.796,A -85,B 0,C 180,E1 -8325.781,E2 -8325.781} C_VEL
LIN {X 0,Y 453.476,Z 661.807,A -85,B 0,C 180,E1 -8328.21,E2 -8328.21} C_VEL
LIN {X 0,Y 453.51,Z 661.809,A -85,B 0,C 180,E1 -8330.791,E2 -8330.791} C_VEL
LIN {X 0,Y 453.465,Z 661.901,A -85,B 0,C 180,E1 -8333.781,E2 -8333.781} C_VEL
LIN {X 0,Y 454.49,Z 665.663,A -85,B 0,C 180,E1 -8334.628,E2 -8334.628} C_VEL
LIN {X 0,Y 457.472,Z 677.082,A -85,B 0,C 180,E1 -8336.951,E2 -8336.951} C_VEL
LIN {X 0,Y 459.753,Z 687.073,A -85,B 0,C 180,E1 -8338.875,E2 -8338.875} C_VEL
LIN {X 0,Y 459.539,Z 693.053,A -85,B 0,C 180,E1 -8339.865,E2 -8339.865} C_VEL
LIN {X 0,Y 466.262,Z 720.448,A -85,B 0,C 180,E1 -8340.844,E2 -8340.844} C_VEL
LIN {X 0,Y 467.453,Z 725.446,A -85,B 0,C 180,E1 -8341.01,E2 -8341.01} C_VEL
LIN {X 0,Y 464.838,Z 894.978,A -85,B 0,C 180,E1 -8343.75,E2 -8343.75} C_VEL
LIN {X 0,Y 464.342,Z 907.32,A -85,B 0,C 180,E1 -8344.026,E2 -8344.026} C_VEL
LIN {X 0,Y 463.705,Z 920.661,A -85,B 0,C 180,E1 -8344.439,E2 -8344.439} C_VEL
LIN {X 0,Y 462.971,Z 933.785,A -85,B 0,C 180,E1 -8344.967,E2 -8344.967} C_VEL
LIN {X 0,Y 462.169,Z 945.175,A -85,B 0,C 180,E1 -8345.521,E2 -8345.521} C_VEL
LIN {X 0,Y 461.207,Z 958.34,A -85,B 0,C 180,E1 -8346.297,E2 -8346.297} C_VEL
LIN {X 0,Y 460.229,Z 969.723,A -85,B 0,C 180,E1 -8347.083,E2 -8347.083} C_VEL
LIN {X 0,Y 459.153,Z 982.165,A -85,B 0,C 180,E1 -8348.094,E2 -8348.094} C_VEL
LIN {X 0,Y 458.149,Z 992.971,A -85,B 0,C 180,E1 -8349.106,E2 -8349.106} C_VEL
LIN {X 0,Y 457.086,Z 1003.473,A -85,B 0,C 180,E1 -8350.229,E2 -8350.229} C_VEL
LIN {X 0,Y 456.275,Z 1012.749,A -85,B 0,C 180,E1 -8351.361,E2 -8351.361} C_VEL
LIN {X 0,Y 455.413,Z 1022.487,A -85,B 0,C 180,E1 -8352.719,E2 -8352.719} C_VEL
LIN {X 0,Y 454.693,Z 1031.014,A -85,B 0,C 180,E1 -8354.077,E2 -8354.077} C_VEL
LIN {X 0,Y 453.954,Z 1039.614,A -85,B 0,C 180,E1 -8355.658,E2 -8355.658} C_VEL
LIN {X 0,Y 453.536,Z 1046.045,A -85,B 0,C 180,E1 -8357.016,E2 -8357.016} C_VEL
LIN {X 0,Y 453.081,Z 1053.301,A -85,B 0,C 180,E1 -8358.82,E2 -8358.82} C_VEL
LIN {X 0,Y 452.788,Z 1057.946,A -85,B 0,C 180,E1 -8360.17,E2 -8360.17} C_VEL
LIN {X 0,Y 452.636,Z 1063.036,A -85,B 0,C 180,E1 -8361.967,E2 -8361.967} C_VEL
LIN {X 0,Y 452.561,Z 1067.025,A -85,B 0,C 180,E1 -8363.759,E2 -8363.759} C_VEL
LIN {X 0,Y 452.441,Z 1069.969,A -85,B 0,C 180,E1 -8365.546,E2 -8365.546} C_VEL
LIN {X 0,Y 452.433,Z 1071.15,A -85,B 0,C 180,E1 -8366.438,E2 -8366.438} C_VEL
LIN {X 0,Y 452.427,Z 1072.611,A -85,B 0,C 180,E1 -8368.22,E2 -8368.22} C_VEL
LIN {X 0,Y 452.43,Z 1073.095,A -85,B 0,C 180,E1 -8370,E2 -8370} C_VEL
LIN {X 0,Y 452.427,Z 1072.611,A -85,B 0,C 180,E1 -8371.78,E2 -8371.78} C_VEL
LIN {X 0,Y 452.433,Z 1071.15,A -85,B 0,C 180,E1 -8373.562,E2 -8373.562} C_VEL
LIN {X 0,Y 452.501,Z 1068.693,A -85,B 0,C 180,E1 -8375.347,E2 -8375.347} C_VEL
LIN {X 0,Y 452.641,Z 1064.123,A -85,B 0,C 180,E1 -8377.584,E2 -8377.584} C_VEL
LIN {X 0,Y 452.709,Z 1060.64,A -85,B 0,C 180,E1 -8378.931,E2 -8378.931} C_VEL
LIN {X 0,Y 452.983,Z 1054.921,A -85,B 0,C 180,E1 -8380.73,E2 -8380.73} C_VEL
LIN {X 0,Y 453.301,Z 1050.057,A -85,B 0,C 180,E1 -8382.036,E2 -8382.036} C_VEL
LIN {X 0,Y 453.804,Z 1041.836,A -85,B 0,C 180,E1 -8383.889,E2 -8383.889} C_VEL
LIN {X 0,Y 454.347,Z 1034.853,A -85,B 0,C 180,E1 -8385.245,E2 -8385.245} C_VEL
LIN {X 0,Y 454.979,Z 1026.919,A -85,B 0,C 180,E1 -8386.599,E2 -8386.599} C_VEL
LIN {X 0,Y 455.808,Z 1017.767,A -85,B 0,C 180,E1 -8387.961,E2 -8387.961} C_VEL
LIN {X 0,Y 456.603,Z 1009.196,A -85,B 0,C 180,E1 -8389.091,E2 -8389.091} C_VEL
